LIN {X 0,Y 626.44,Z 347.198,A -85,B 0,C 180,E1 29853.409,E2 29853.409} C_VEL
LIN {X 0,Y 625.043,Z 344.117,A -85,B 0,C 180,E1 29853.056,E2 29853.056} C_VEL
LIN {X 0,Y 624.945,Z 343.42,A -85,B 0,C 180,E1 29852.768,E2 29852.768} C_VEL
LIN {X 0,Y 624.921,Z 343.391,A -85,B 0,C 180,E1 29849.587,E2 29849.587} C_VEL
LIN {X 0,Y 624.985,Z 343.634,A -85,B 0,C 180,E1 29846.589,E2 29846.589} C_VEL
LIN {X 0,Y 626.32,Z 346.962,A -85,B 0,C 180,E1 29846.03,E2 29846.03} C_VEL
LIN {X 0,Y 627.286,Z 348.589,A -85,B 0,C 180,E1 29845.758,E2 29845.758} C_VEL
LIN {X 0,Y 631.043,Z 356.586,A -85,B 0,C 180,E1 29844.666,E2 29844.666} C_VEL
LIN {X 0,Y 636.482,Z 369.43,A -85,B 0,C 180,E1 29843.235,E2 29843.235} C_VEL
LIN {X 0,Y 643.968,Z 387.871,A -85,B 0,C 180,E1 29841.491,E2 29841.491} C_VEL
LIN {X 0,Y 650.226,Z 398.532,A -85,B 0,C 180,E1 29840.459,E2 29840.459} C_VEL
LIN {X 0,Y 650.452,Z 412.85,A -85,B 0,C 180,E1 29839.657,E2 29839.657} C_VEL
LIN {X 0,Y 655.73,Z 440.789,A -85,B 0,C 180,E1 29838.782,E2 29838.782} C_VEL
LIN {X 0,Y 660.63,Z 462.04,A -85,B 0,C 180,E1 29838.099,E2 29838.099} C_VEL
LIN {X 0,Y 658.56,Z 625.386,A -85,B 0,C 180,E1 29835.964,E2 29835.964} C_VEL
LIN {X 0,Y 654.313,Z 847.674,A -85,B 0,C 180,E1 29832.989,E2 29832.989} C_VEL
LIN {X 0,Y 653.026,Z 907.79,A -85,B 0,C 180,E1 29832.173,E2 29832.173} C_VEL
LIN {X 0,Y 651.72,Z 936.587,A -85,B 0,C 180,E1 29831.618,E2 29831.618} C_VEL
LIN {X 0,Y 650.342,Z 959.946,A -85,B 0,C 180,E1 29831.02,E2 29831.02} C_VEL
LIN {X 0,Y 648.895,Z 981.108,A -85,B 0,C 180,E1 29830.358,E2 29830.358} C_VEL
LIN {X 0,Y 647.293,Z 1002.373,A -85,B 0,C 180,E1 29829.572,E2 29829.572} C_VEL
LIN {X 0,Y 645.185,Z 1027.649,A -85,B 0,C 180,E1 29828.479,E2 29828.479} C_VEL
LIN {X 0,Y 642.948,Z 1051.037,A -85,B 0,C 180,E1 29827.281,E2 29827.281} C_VEL
LIN {X 0,Y 640.981,Z 1070.815,A -85,B 0,C 180,E1 29826.132,E2 29826.132} C_VEL
LIN {X 0,Y 639.019,Z 1089.996,A -85,B 0,C 180,E1 29824.883,E2 29824.883} C_VEL
LIN {X 0,Y 636.733,Z 1111.873,A -85,B 0,C 180,E1 29823.287,E2 29823.287} C_VEL
LIN {X 0,Y 634.481,Z 1133.139,A -85,B 0,C 180,E1 29821.507,E2 29821.507} C_VEL
LIN {X 0,Y 632.771,Z 1149.796,A -85,B 0,C 180,E1 29819.956,E2 29819.956} C_VEL
LIN {X 0,Y 631.114,Z 1166.381,A -85,B 0,C 180,E1 29818.25,E2 29818.25} C_VEL
LIN {X 0,Y 629.253,Z 1185.743,A -85,B 0,C 180,E1 29816.012,E2 29816.012} C_VEL
LIN {X 0,Y 627.941,Z 1200.693,A -85,B 0,C 180,E1 29814.056,E2 29814.056} C_VEL
LIN {X 0,Y 626.836,Z 1214.647,A -85,B 0,C 180,E1 29812.015,E2 29812.015} C_VEL
LIN {X 0,Y 625.791,Z 1229.67,A -85,B 0,C 180,E1 29809.508,E2 29809.508} C_VEL
LIN {X 0,Y 625.132,Z 1240.614,A -85,B 0,C 180,E1 29807.403,E2 29807.403} C_VEL
LIN {X 0,Y 624.666,Z 1249.714,A -85,B 0,C 180,E1 29805.409,E2 29805.409} C_VEL
LIN {X 0,Y 624.334,Z 1258.281,A -85,B 0,C 180,E1 29803.239,E2 29803.239} C_VEL
LIN {X 0,Y 624.09,Z 1266.776,A -85,B 0,C 180,E1 29800.617,E2 29800.617} C_VEL
LIN {X 0,Y 623.98,Z 1272.734,A -85,B 0,C 180,E1 29798.292,E2 29798.292} C_VEL
LIN {X 0,Y 623.933,Z 1277.189,A -85,B 0,C 180,E1 29795.979,E2 29795.979} C_VEL
LIN {X 0,Y 623.912,Z 1280.336,A -85,B 0,C 180,E1 29793.491,E2 29793.491} C_VEL
LIN {X 0,Y 623.889,Z 1281.714,A -85,B 0,C 180,E1 29791.194,E2 29791.194} C_VEL
LIN {X 0,Y 623.864,Z 1281.827,A -85,B 0,C 180,E1 29789.265,E2 29789.265} C_VEL
LIN {X 0,Y 623.908,Z 1280.947,A -85,B 0,C 180,E1 29787.336,E2 29787.336} C_VEL
LIN {X 0,Y 623.916,Z 1278.899,A -85,B 0,C 180,E1 29785.22,E2 29785.22} C_VEL
LIN {X 0,Y 623.954,Z 1275.078,A -85,B 0,C 180,E1 29782.82,E2 29782.82} C_VEL
LIN {X 0,Y 623.985,Z 1269.837,A -85,B 0,C 180,E1 29780.5,E2 29780.5} C_VEL
LIN {X 0,Y 624.176,Z 1263.356,A -85,B 0,C 180,E1 29778.262,E2 29778.262} C_VEL
LIN {X 0,Y 624.361,Z 1256.514,A -85,B 0,C 180,E1 29776.29,E2 29776.29} C_VEL
LIN {X 0,Y 624.701,Z 1248.901,A -85,B 0,C 180,E1 29774.401,E2 29774.401} C_VEL
LIN {X 0,Y 625.202,Z 1239.22,A -85,B 0,C 180,E1 29772.31,E2 29772.31} C_VEL
LIN {X 0,Y 626.035,Z 1225.878,A -85,B 0,C 180,E1 29769.819,E2 29769.819} C_VEL
LIN {X 0,Y 626.999,Z 1212.519,A -85,B 0,C 180,E1 29767.66,E2 29767.66} C_VEL
LIN {X 0,Y 628.138,Z 1198.567,A -85,B 0,C 180,E1 29765.652,E2 29765.652} C_VEL
LIN {X 0,Y 629.787,Z 1180.067,A -85,B 0,C 180,E1 29763.301,E2 29763.301} C_VEL
LIN {X 0,Y 631.389,Z 1163.378,A -85,B 0,C 180,E1 29761.429,E2 29761.429} C_VEL
LIN {X 0,Y 633.123,Z 1146.246,A -85,B 0,C 180,E1 29759.697,E2 29759.697} C_VEL
LIN {X 0,Y 635.507,Z 1123.476,A -85,B 0,C 180,E1 29757.66,E2 29757.66} C_VEL
LIN {X 0,Y 637.417,Z 1105.296,A -85,B 0,C 180,E1 29756.22,E2 29756.22} C_VEL
LIN {X 0,Y 639.321,Z 1087.049,A -85,B 0,C 180,E1 29754.917,E2 29754.917} C_VEL
LIN {X 0,Y 641.405,Z 1066.751,A -85,B 0,C 180,E1 29753.619,E2 29753.619} C_VEL
LIN {X 0,Y 643.914,Z 1040.714,A -85,B 0,C 180,E1 29752.167,E2 29752.167} C_VEL
LIN {X 0,Y 645.879,Z 1018.721,A -85,B 0,C 180,E1 29751.116,E2 29751.116} C_VEL
LIN {X 0,Y 647.601,Z 998.037,A -85,B 0,C 180,E1 29750.256,E2 29750.256} C_VEL
LIN {X 0,Y 649.274,Z 975.928,A -85,B 0,C 180,E1 29749.468,E2 29749.468} C_VEL
LIN {X 0,Y 651.08,Z 948.454,A -85,B 0,C 180,E1 29748.665,E2 29748.665} C_VEL
LIN {X 0,Y 652.353,Z 923.49,A -85,B 0,C 180,E1 29748.107,E2 29748.107} C_VEL
LIN {X 0,Y 653.236,Z 900.801,A -85,B 0,C 180,E1 29747.723,E2 29747.723} C_VEL
LIN {X 0,Y 657.429,Z 682.384,A -85,B 0,C 180,E1 29744.806,E2 29744.806} C_VEL
LIN {X 0,Y 661.107,Z 486.103,A -85,B 0,C 180,E1 29742.148,E2 29742.148} C_VEL
LIN {X 0,Y 661.403,Z 460.724,A -85,B 0,C 180,E1 29741.783,E2 29741.783} C_VEL
LIN {X 0,Y 653.875,Z 423.501,A -85,B 0,C 180,E1 29740.419,E2 29740.419} C_VEL
LIN {X 0,Y 655.004,Z 402.248,A -85,B 0,C 180,E1 29739.014,E2 29739.014} C_VEL
LIN {X 0,Y 643.082,Z 378.276,A -85,B 0,C 180,E1 29735.996,E2 29735.996} C_VEL
LIN {X 0,Y 636.424,Z 365.479,A -85,B 0,C 180,E1 29734.226,E2 29734.226} C_VEL
LIN {X 0,Y 631.891,Z 356.934,A -85,B 0,C 180,E1 29732.98,E2 29732.98} C_VEL
LIN {X 0,Y 629.323,Z 352.257,A -85,B 0,C 180,E1 29732.266,E2 29732.266} C_VEL
LIN {X 0,Y 626.8,Z 347.598,A -85,B 0,C 180,E1 29731.55,E2 29731.55} C_VEL
LIN {X 0,Y 625.074,Z 344.123,A -85,B 0,C 180,E1 29731.003,E2 29731.003} C_VEL
LIN {X 0,Y 624.943,Z 343.458,A -85,B 0,C 180,E1 29730.776,E2 29730.776} C_VEL
LIN {X 0,Y 624.946,Z 343.386,A -85,B 0,C 180,E1 29727.645,E2 29727.645} C_VEL
LIN {X 0,Y 624.927,Z 343.382,A -85,B 0,C 180,E1 29724.482,E2 29724.482} C_VEL
LIN {X 0,Y 624.945,Z 343.377,A -85,B 0,C 180,E1 29721.383,E2 29721.383} C_VEL
LIN {X 0,Y 624.924,Z 343.376,A -85,B 0,C 180,E1 29718.277,E2 29718.277} C_VEL
LIN {X 0,Y 624.945,Z 343.375,A -85,B 0,C 180,E1 29715.212,E2 29715.212} C_VEL
LIN {X 0,Y 624.921,Z 343.375,A -85,B 0,C 180,E1 29712.099,E2 29712.099} C_VEL
LIN {X 0,Y 624.947,Z 343.377,A -85,B 0,C 180,E1 29709.021,E2 29709.021} C_VEL
LIN {X 0,Y 624.919,Z 343.378,A -85,B 0,C 180,E1 29705.97,E2 29705.97} C_VEL
LIN {X 0,Y 624.949,Z 343.384,A -85,B 0,C 180,E1 29702.843,E2 29702.843} C_VEL
LIN {X 0,Y 624.916,Z 343.386,A -85,B 0,C 180,E1 29699.725,E2 29699.725} C_VEL
LIN {X 0,Y 624.949,Z 343.382,A -85,B 0,C 180,E1 29696.606,E2 29696.606} C_VEL
LIN {X 0,Y 624.912,Z 343.384,A -85,B 0,C 180,E1 29693.477,E2 29693.477} C_VEL
LIN {X 0,Y 624.952,Z 343.382,A -85,B 0,C 180,E1 29690.422,E2 29690.422} C_VEL
LIN {X 0,Y 624.911,Z 343.386,A -85,B 0,C 180,E1 29687.337,E2 29687.337} C_VEL
LIN {X 0,Y 624.956,Z 343.382,A -85,B 0,C 180,E1 29684.312,E2 29684.312} C_VEL
LIN {X 0,Y 624.91,Z 343.387,A -85,B 0,C 180,E1 29681.239,E2 29681.239} C_VEL
LIN {X 0,Y 624.956,Z 343.381,A -85,B 0,C 180,E1 29678.211,E2 29678.211} C_VEL
LIN {X 0,Y 624.911,Z 343.387,A -85,B 0,C 180,E1 29675.114,E2 29675.114} C_VEL
LIN {X 0,Y 624.957,Z 343.381,A -85,B 0,C 180,E1 29672.025,E2 29672.025} C_VEL
LIN {X 0,Y 624.905,Z 343.387,A -85,B 0,C 180,E1 29668.873,E2 29668.873} C_VEL
LIN {X 0,Y 624.954,Z 343.381,A -85,B 0,C 180,E1 29665.808,E2 29665.808} C_VEL
LIN {X 0,Y 624.9,Z 343.388,A -85,B 0,C 180,E1 29662.668,E2 29662.668} C_VEL
LIN {X 0,Y 624.942,Z 343.381,A -85,B 0,C 180,E1 29659.73,E2 29659.73} C_VEL
LIN {X 0,Y 624.901,Z 343.388,A -85,B 0,C 180,E1 29656.525,E2 29656.525} C_VEL
LIN {X 0,Y 624.938,Z 343.381,A -85,B 0,C 180,E1 29653.548,E2 29653.548} C_VEL
LIN {X 0,Y 624.899,Z 343.389,A -85,B 0,C 180,E1 29650.391,E2 29650.391} C_VEL
LIN {X 0,Y 624.889,Z 343.386,A -85,B 0,C 180,E1 29648.108,E2 29648.108} C_VEL
LIN {X 0,Y 623.91,Z 343.51,A -85,B 0,C 180,E1 29647.401,E2 29647.401} C_VEL
LIN {X 0,Y 617.551,Z 344.298,A -85,B 0,C 180,E1 29645.42,E2 29645.42} C_VEL
LIN {X 0,Y 617.016,Z 344.367,A -85,B 0,C 180,E1 29644.905,E2 29644.905} C_VEL
LIN {X 0,Y 616.947,Z 344.374,A -85,B 0,C 180,E1 29641.869,E2 29641.869} C_VEL
LIN {X 0,Y 617.019,Z 344.364,A -85,B 0,C 180,E1 29638.875,E2 29638.875} C_VEL
LIN {X 0,Y 616.947,Z 344.375,A -85,B 0,C 180,E1 29635.847,E2 29635.847} C_VEL
LIN {X 0,Y 616.991,Z 344.365,A -85,B 0,C 180,E1 29632.888,E2 29632.888} C_VEL
LIN {X 0,Y 616.949,Z 344.379,A -85,B 0,C 180,E1 29629.799,E2 29629.799} C_VEL
LIN {X 0,Y 616.959,Z 344.374,A -85,B 0,C 180,E1 29626.961,E2 29626.961} C_VEL
LIN {X 0,Y 616.952,Z 344.379,A -85,B 0,C 180,E1 29623.687,E2 29623.687} C_VEL
LIN {X 0,Y 616.944,Z 344.379,A -85,B 0,C 180,E1 29620.931,E2 29620.931} C_VEL
LIN {X 0,Y 616.968,Z 344.374,A -85,B 0,C 180,E1 29617.73,E2 29617.73} C_VEL
LIN {X 0,Y 616.931,Z 344.373,A -85,B 0,C 180,E1 29614.928,E2 29614.928} C_VEL
LIN {X 0,Y 617.003,Z 344.374,A -85,B 0,C 180,E1 29611.857,E2 29611.857} C_VEL
LIN {X 0,Y 616.929,Z 344.382,A -85,B 0,C 180,E1 29608.979,E2 29608.979} C_VEL
LIN {X 0,Y 616.97,Z 344.359,A -85,B 0,C 180,E1 29606.097,E2 29606.097} C_VEL
LIN {X 0,Y 616.931,Z 344.354,A -85,B 0,C 180,E1 29603.018,E2 29603.018} C_VEL
LIN {X 0,Y 616.926,Z 344.371,A -85,B 0,C 180,E1 29600.39,E2 29600.39} C_VEL
LIN {X 0,Y 617.025,Z 344.571,A -85,B 0,C 180,E1 29597.601,E2 29597.601} C_VEL
LIN {X 0,Y 617.381,Z 346.03,A -85,B 0,C 180,E1 29597.395,E2 29597.395} C_VEL
LIN {X 0,Y 619.284,Z 349.081,A -85,B 0,C 180,E1 29597.102,E2 29597.102} C_VEL
LIN {X 0,Y 621.278,Z 350.95,A -85,B 0,C 180,E1 29596.83,E2 29596.83} C_VEL
LIN {X 0,Y 623.786,Z 354.703,A -85,B 0,C 180,E1 29596.466,E2 29596.466} C_VEL
LIN {X 0,Y 625.81,Z 356.86,A -85,B 0,C 180,E1 29596.193,E2 29596.193} C_VEL
LIN {X 0,Y 629.122,Z 361.131,A -85,B 0,C 180,E1 29595.739,E2 29595.739} C_VEL
LIN {X 0,Y 633.273,Z 366.632,A -85,B 0,C 180,E1 29595.18,E2 29595.18} C_VEL
LIN {X 0,Y 649.293,Z 388.598,A -85,B 0,C 180,E1 29593.148,E2 29593.148} C_VEL
LIN {X 0,Y 654.652,Z 396.391,A -85,B 0,C 180,E1 29592.508,E2 29592.508} C_VEL
LIN {X 0,Y 650.14,Z 613.265,A -85,B 0,C 180,E1 29589.557,E2 29589.557} C_VEL
LIN {X 0,Y 647.14,Z 757.621,A -85,B 0,C 180,E1 29587.612,E2 29587.612} C_VEL
LIN {X 0,Y 645.877,Z 783.784,A -85,B 0,C 180,E1 29587.113,E2 29587.113} C_VEL
LIN {X 0,Y 644.236,Z 810.568,A -85,B 0,C 180,E1 29586.432,E2 29586.432} C_VEL
LIN {X 0,Y 642.332,Z 836.613,A -85,B 0,C 180,E1 29585.595,E2 29585.595} C_VEL
LIN {X 0,Y 640.2,Z 862.261,A -85,B 0,C 180,E1 29584.589,E2 29584.589} C_VEL
LIN {X 0,Y 637.88,Z 886.313,A -85,B 0,C 180,E1 29583.466,E2 29583.466} C_VEL
LIN {X 0,Y 635.242,Z 911.914,A -85,B 0,C 180,E1 29582.073,E2 29582.073} C_VEL
LIN {X 0,Y 632.667,Z 935.913,A -85,B 0,C 180,E1 29580.555,E2 29580.555} C_VEL
LIN {X 0,Y 630.387,Z 956.418,A -85,B 0,C 180,E1 29579.076,E2 29579.076} C_VEL
LIN {X 0,Y 627.823,Z 978.962,A -85,B 0,C 180,E1 29577.237,E2 29577.237} C_VEL
LIN {X 0,Y 625.456,Z 1000.26,A -85,B 0,C 180,E1 29575.257,E2 29575.257} C_VEL
LIN {X 0,Y 623.342,Z 1020.045,A -85,B 0,C 180,E1 29573.172,E2 29573.172} C_VEL
LIN {X 0,Y 621.513,Z 1038.014,A -85,B 0,C 180,E1 29571.021,E2 29571.021} C_VEL
LIN {X 0,Y 619.972,Z 1054.397,A -85,B 0,C 180,E1 29568.807,E2 29568.807} C_VEL
LIN {X 0,Y 618.665,Z 1070.031,A -85,B 0,C 180,E1 29566.391,E2 29566.391} C_VEL
LIN {X 0,Y 617.768,Z 1082.311,A -85,B 0,C 180,E1 29564.235,E2 29564.235} C_VEL
LIN {X 0,Y 617.026,Z 1093.97,A -85,B 0,C 180,E1 29561.886,E2 29561.886} C_VEL
LIN {X 0,Y 616.526,Z 1104.735,A -85,B 0,C 180,E1 29559.322,E2 29559.322} C_VEL
LIN {X 0,Y 616.199,Z 1112.49,A -85,B 0,C 180,E1 29557.131,E2 29557.131} C_VEL
LIN {X 0,Y 616.046,Z 1119.459,A -85,B 0,C 180,E1 29554.73,E2 29554.73} C_VEL
LIN {X 0,Y 615.934,Z 1124.777,A -85,B 0,C 180,E1 29552.393,E2 29552.393} C_VEL
LIN {X 0,Y 615.929,Z 1128.644,A -85,B 0,C 180,E1 29550,E2 29550} C_VEL
LIN {X 0,Y 615.888,Z 1131.051,A -85,B 0,C 180,E1 29547.574,E2 29547.574} C_VEL
LIN {X 0,Y 615.901,Z 1131.941,A -85,B 0,C 180,E1 29545.276,E2 29545.276} C_VEL
LIN {X 0,Y 615.865,Z 1131.328,A -85,B 0,C 180,E1 29542.756,E2 29542.756} C_VEL
LIN {X 0,Y 615.915,Z 1129.328,A -85,B 0,C 180,E1 29540.428,E2 29540.428} C_VEL
LIN {X 0,Y 615.948,Z 1125.598,A -85,B 0,C 180,E1 29537.962,E2 29537.962} C_VEL
LIN {X 0,Y 616.037,Z 1120.12,A -85,B 0,C 180,E1 29535.438,E2 29535.438} C_VEL
LIN {X 0,Y 616.205,Z 1113.002,A -85,B 0,C 180,E1 29532.94,E2 29532.94} C_VEL
LIN {X 0,Y 616.487,Z 1105.704,A -85,B 0,C 180,E1 29530.844,E2 29530.844} C_VEL
LIN {X 0,Y 616.969,Z 1095.624,A -85,B 0,C 180,E1 29528.387,E2 29528.387} C_VEL
LIN {X 0,Y 617.681,Z 1083.75,A -85,B 0,C 180,E1 29525.947,E2 29525.947} C_VEL
LIN {X 0,Y 618.592,Z 1071.179,A -85,B 0,C 180,E1 29523.707,E2 29523.707} C_VEL
LIN {X 0,Y 619.811,Z 1056.349,A -85,B 0,C 180,E1 29521.387,E2 29521.387} C_VEL
LIN {X 0,Y 621.372,Z 1039.468,A -85,B 0,C 180,E1 29519.078,E2 29519.078} C_VEL
LIN {X 0,Y 623.025,Z 1022.847,A -85,B 0,C 180,E1 29517.056,E2 29517.056} C_VEL
LIN {X 0,Y 625.243,Z 1002.388,A -85,B 0,C 180,E1 29514.862,E2 29514.862} C_VEL
LIN {X 0,Y 627.462,Z 982.118,A -85,B 0,C 180,E1 29512.952,E2 29512.952} C_VEL
LIN {X 0,Y 630.054,Z 959.257,A -85,B 0,C 180,E1 29511.053,E2 29511.053} C_VEL
LIN {X 0,Y 632.554,Z 937.101,A -85,B 0,C 180,E1 29509.434,E2 29509.434} C_VEL
LIN {X 0,Y 635.206,Z 912.533,A -85,B 0,C 180,E1 29507.869,E2 29507.869} C_VEL
LIN {X 0,Y 637.696,Z 888.159,A -85,B 0,C 180,E1 29506.535,E2 29506.535} C_VEL
LIN {X 0,Y 640.033,Z 863.672,A -85,B 0,C 180,E1 29505.386,E2 29505.386} C_VEL
LIN {X 0,Y 642.204,Z 838.307,A -85,B 0,C 180,E1 29504.374,E2 29504.374} C_VEL
LIN {X 0,Y 644.064,Z 812.942,A -85,B 0,C 180,E1 29503.547,E2 29503.547} C_VEL
LIN {X 0,Y 645.778,Z 785.479,A -85,B 0,C 180,E1 29502.836,E2 29502.836} C_VEL
LIN {X 0,Y 647.033,Z 760.107,A -85,B 0,C 180,E1 29502.34,E2 29502.34} C_VEL
LIN {X 0,Y 648.218,Z 710.458,A -85,B 0,C 180,E1 29501.653,E2 29501.653} C_VEL
LIN {X 0,Y 652.209,Z 504.112,A -85,B 0,C 180,E1 29498.893,E2 29498.893} C_VEL
LIN {X 0,Y 654.095,Z 395.736,A -85,B 0,C 180,E1 29497.413,E2 29497.413} C_VEL
LIN {X 0,Y 639.586,Z 375.63,A -85,B 0,C 180,E1 29495.674,E2 29495.674} C_VEL
LIN {X 0,Y 632.819,Z 366.077,A -85,B 0,C 180,E1 29494.712,E2 29494.712} C_VEL
LIN {X 0,Y 629.184,Z 361.107,A -85,B 0,C 180,E1 29494.145,E2 29494.145} C_VEL
LIN {X 0,Y 626.323,Z 356.874,A -85,B 0,C 180,E1 29493.641,E2 29493.641} C_VEL
LIN {X 0,Y 622.996,Z 353.334,A -85,B 0,C 180,E1 29493.05,E2 29493.05} C_VEL
LIN {X 0,Y 621.527,Z 350.643,A -85,B 0,C 180,E1 29492.726,E2 29492.726} C_VEL
LIN {X 0,Y 618.454,Z 348.053,A -85,B 0,C 180,E1 29492.073,E2 29492.073} C_VEL
LIN {X 0,Y 617.11,Z 345.139,A -85,B 0,C 180,E1 29491.618,E2 29491.618} C_VEL
LIN {X 0,Y 616.977,Z 344.413,A -85,B 0,C 180,E1 29491.228,E2 29491.228} C_VEL
LIN {X 0,Y 617.014,Z 344.376,A -85,B 0,C 180,E1 29488.11,E2 29488.11} C_VEL
LIN {X 0,Y 617.06,Z 344.812,A -85,B 0,C 180,E1 29487.674,E2 29487.674} C_VEL
LIN {X 0,Y 618.456,Z 348.097,A -85,B 0,C 180,E1 29486.986,E2 29486.986} C_VEL
LIN {X 0,Y 619.613,Z 349.9,A -85,B 0,C 180,E1 29486.613,E2 29486.613} C_VEL
LIN {X 0,Y 622.023,Z 355.115,A -85,B 0,C 180,E1 29485.763,E2 29485.763} C_VEL
LIN {X 0,Y 625.43,Z 362.431,A -85,B 0,C 180,E1 29484.75,E2 29484.75} C_VEL
LIN {X 0,Y 630.385,Z 374.351,A -85,B 0,C 180,E1 29483.388,E2 29483.388} C_VEL
LIN {X 0,Y 637.71,Z 392.65,A -85,B 0,C 180,E1 29481.618,E2 29481.618} C_VEL
LIN {X 0,Y 643.308,Z 402.169,A -85,B 0,C 180,E1 29480.671,E2 29480.671} C_VEL
LIN {X 0,Y 643.497,Z 407.96,A -85,B 0,C 180,E1 29480.361,E2 29480.361} C_VEL
LIN {X 0,Y 650.125,Z 444.426,A -85,B 0,C 180,E1 29479.171,E2 29479.171} C_VEL
LIN {X 0,Y 654.533,Z 463.978,A -85,B 0,C 180,E1 29478.531,E2 29478.531} C_VEL
LIN {X 0,Y 652.544,Z 612.386,A -85,B 0,C 180,E1 29476.579,E2 29476.579} C_VEL
LIN {X 0,Y 651.281,Z 707.38,A -85,B 0,C 180,E1 29475.355,E2 29475.355} C_VEL
LIN {X 0,Y 647.193,Z 904.317,A -85,B 0,C 180,E1 29472.703,E2 29472.703} C_VEL
LIN {X 0,Y 646.07,Z 930.59,A -85,B 0,C 180,E1 29472.23,E2 29472.23} C_VEL
LIN {X 0,Y 644.42,Z 957.585,A -85,B 0,C 180,E1 29471.56,E2 29471.56} C_VEL
LIN {X 0,Y 642.878,Z 979.062,A -85,B 0,C 180,E1 29470.896,E2 29470.896} C_VEL
LIN {X 0,Y 641.217,Z 999.571,A -85,B 0,C 180,E1 29470.15,E2 29470.15} C_VEL
LIN {X 0,Y 639.315,Z 1020.973,A -85,B 0,C 180,E1 29469.244,E2 29469.244} C_VEL
LIN {X 0,Y 636.881,Z 1046.532,A -85,B 0,C 180,E1 29467.983,E2 29467.983} C_VEL
LIN {X 0,Y 634.478,Z 1069.189,A -85,B 0,C 180,E1 29466.674,E2 29466.674} C_VEL
LIN {X 0,Y 632.44,Z 1087.789,A -85,B 0,C 180,E1 29465.466,E2 29465.466} C_VEL
LIN {X 0,Y 630.425,Z 1105.899,A -85,B 0,C 180,E1 29464.156,E2 29464.156} C_VEL
LIN {X 0,Y 628.076,Z 1126.929,A -85,B 0,C 180,E1 29462.461,E2 29462.461} C_VEL
LIN {X 0,Y 625.702,Z 1147.856,A -85,B 0,C 180,E1 29460.532,E2 29460.532} C_VEL
LIN {X 0,Y 623.918,Z 1164.304,A -85,B 0,C 180,E1 29458.841,E2 29458.841} C_VEL
LIN {X 0,Y 622.05,Z 1182.6,A -85,B 0,C 180,E1 29456.748,E2 29456.748} C_VEL
LIN {X 0,Y 620.377,Z 1199.99,A -85,B 0,C 180,E1 29454.47,E2 29454.47} C_VEL
LIN {X 0,Y 619.154,Z 1214.01,A -85,B 0,C 180,E1 29452.403,E2 29452.403} C_VEL
LIN {X 0,Y 618.004,Z 1229.149,A -85,B 0,C 180,E1 29449.862,E2 29449.862} C_VEL
LIN {X 0,Y 617.245,Z 1240.616,A -85,B 0,C 180,E1 29447.633,E2 29447.633} C_VEL
LIN {X 0,Y 616.719,Z 1250.117,A -85,B 0,C 180,E1 29445.516,E2 29445.516} C_VEL
LIN {X 0,Y 616.351,Z 1259.339,A -85,B 0,C 180,E1 29443.127,E2 29443.127} C_VEL
LIN {X 0,Y 616.099,Z 1267.033,A -85,B 0,C 180,E1 29440.662,E2 29440.662} C_VEL
LIN {X 0,Y 615.994,Z 1272.731,A -85,B 0,C 180,E1 29438.4,E2 29438.4} C_VEL
LIN {X 0,Y 615.934,Z 1277.337,A -85,B 0,C 180,E1 29435.963,E2 29435.963} C_VEL
LIN {X 0,Y 615.911,Z 1280.404,A -85,B 0,C 180,E1 29433.444,E2 29433.444} C_VEL
LIN {X 0,Y 615.89,Z 1281.714,A -85,B 0,C 180,E1 29431.209,E2 29431.209} C_VEL
LIN {X 0,Y 615.864,Z 1281.827,A -85,B 0,C 180,E1 29429.256,E2 29429.256} C_VEL
LIN {X 0,Y 615.908,Z 1280.947,A -85,B 0,C 180,E1 29427.302,E2 29427.302} C_VEL
LIN {X 0,Y 615.916,Z 1279.009,A -85,B 0,C 180,E1 29425.251,E2 29425.251} C_VEL
LIN {X 0,Y 615.956,Z 1275.25,A -85,B 0,C 180,E1 29422.82,E2 29422.82} C_VEL
LIN {X 0,Y 616.001,Z 1269.837,A -85,B 0,C 180,E1 29420.376,E2 29420.376} C_VEL
LIN {X 0,Y 616.197,Z 1263.306,A -85,B 0,C 180,E1 29418.092,E2 29418.092} C_VEL
LIN {X 0,Y 616.406,Z 1256.513,A -85,B 0,C 180,E1 29416.109,E2 29416.109} C_VEL
LIN {X 0,Y 616.785,Z 1248.902,A -85,B 0,C 180,E1 29414.196,E2 29414.196} C_VEL
LIN {X 0,Y 617.314,Z 1239.222,A -85,B 0,C 180,E1 29412.076,E2 29412.076} C_VEL
LIN {X 0,Y 618.227,Z 1225.876,A -85,B 0,C 180,E1 29409.553,E2 29409.553} C_VEL
LIN {X 0,Y 619.255,Z 1212.741,A -85,B 0,C 180,E1 29407.401,E2 29407.401} C_VEL
LIN {X 0,Y 620.507,Z 1198.569,A -85,B 0,C 180,E1 29405.333,E2 29405.333} C_VEL
LIN {X 0,Y 622.307,Z 1180.065,A -85,B 0,C 180,E1 29402.954,E2 29402.954} C_VEL
LIN {X 0,Y 624.01,Z 1163.377,A -85,B 0,C 180,E1 29401.059,E2 29401.059} C_VEL
LIN {X 0,Y 625.88,Z 1146.243,A -85,B 0,C 180,E1 29399.308,E2 29399.308} C_VEL
LIN {X 0,Y 628.451,Z 1123.477,A -85,B 0,C 180,E1 29397.252,E2 29397.252} C_VEL
LIN {X 0,Y 630.495,Z 1105.226,A -85,B 0,C 180,E1 29395.793,E2 29395.793} C_VEL
LIN {X 0,Y 632.487,Z 1087.352,A -85,B 0,C 180,E1 29394.504,E2 29394.504} C_VEL
LIN {X 0,Y 634.565,Z 1068.371,A -85,B 0,C 180,E1 29393.275,E2 29393.275} C_VEL
LIN {X 0,Y 637.07,Z 1044.692,A -85,B 0,C 180,E1 29391.916,E2 29391.916} C_VEL
LIN {X 0,Y 639.415,Z 1019.848,A -85,B 0,C 180,E1 29390.705,E2 29390.705} C_VEL
LIN {X 0,Y 641.277,Z 998.805,A -85,B 0,C 180,E1 29389.82,E2 29389.82} C_VEL
LIN {X 0,Y 643.002,Z 977.405,A -85,B 0,C 180,E1 29389.047,E2 29389.047} C_VEL
LIN {X 0,Y 644.867,Z 951.337,A -85,B 0,C 180,E1 29388.264,E2 29388.264} C_VEL
LIN {X 0,Y 646.329,Z 924.602,A -85,B 0,C 180,E1 29387.653,E2 29387.653} C_VEL
LIN {X 0,Y 647.275,Z 901.947,A -85,B 0,C 180,E1 29387.262,E2 29387.262} C_VEL
LIN {X 0,Y 651.587,Z 691.755,A -85,B 0,C 180,E1 29384.433,E2 29384.433} C_VEL
LIN {X 0,Y 655.567,Z 485.945,A -85,B 0,C 180,E1 29381.639,E2 29381.639} C_VEL
LIN {X 0,Y 655.86,Z 462.778,A -85,B 0,C 180,E1 29381.303,E2 29381.303} C_VEL
LIN {X 0,Y 647.915,Z 422.962,A -85,B 0,C 180,E1 29379.825,E2 29379.825} C_VEL
LIN {X 0,Y 648.846,Z 406.53,A -85,B 0,C 180,E1 29378.731,E2 29378.731} C_VEL
LIN {X 0,Y 636.194,Z 380.875,A -85,B 0,C 180,E1 29375.447,E2 29375.447} C_VEL
LIN {X 0,Y 626.696,Z 362.853,A -85,B 0,C 180,E1 29372.852,E2 29372.852} C_VEL
LIN {X 0,Y 621.626,Z 353.526,A -85,B 0,C 180,E1 29371.41,E2 29371.41} C_VEL
LIN {X 0,Y 619.174,Z 348.965,A -85,B 0,C 180,E1 29370.684,E2 29370.684} C_VEL
LIN {X 0,Y 617.266,Z 345.616,A -85,B 0,C 180,E1 29370.118,E2 29370.118} C_VEL
LIN {X 0,Y 617.035,Z 344.519,A -85,B 0,C 180,E1 29369.895,E2 29369.895} C_VEL
LIN {X 0,Y 616.994,Z 344.365,A -85,B 0,C 180,E1 29366.673,E2 29366.673} C_VEL
LIN {X 0,Y 617.005,Z 344.362,A -85,B 0,C 180,E1 29363.494,E2 29363.494} C_VEL
LIN {X 0,Y 616.988,Z 344.369,A -85,B 0,C 180,E1 29360.391,E2 29360.391} C_VEL
LIN {X 0,Y 617.006,Z 344.367,A -85,B 0,C 180,E1 29357.251,E2 29357.251} C_VEL
LIN {X 0,Y 616.985,Z 344.375,A -85,B 0,C 180,E1 29354.165,E2 29354.165} C_VEL
LIN {X 0,Y 617.008,Z 344.365,A -85,B 0,C 180,E1 29351.024,E2 29351.024} C_VEL
LIN {X 0,Y 616.98,Z 344.372,A -85,B 0,C 180,E1 29347.918,E2 29347.918} C_VEL
LIN {X 0,Y 617.008,Z 344.36,A -85,B 0,C 180,E1 29344.834,E2 29344.834} C_VEL
LIN {X 0,Y 616.977,Z 344.363,A -85,B 0,C 180,E1 29341.765,E2 29341.765} C_VEL
LIN {X 0,Y 617.011,Z 344.371,A -85,B 0,C 180,E1 29338.7,E2 29338.7} C_VEL
LIN {X 0,Y 616.975,Z 344.372,A -85,B 0,C 180,E1 29335.538,E2 29335.538} C_VEL
LIN {X 0,Y 617.013,Z 344.371,A -85,B 0,C 180,E1 29332.457,E2 29332.457} C_VEL
LIN {X 0,Y 616.972,Z 344.374,A -85,B 0,C 180,E1 29329.353,E2 29329.353} C_VEL
LIN {X 0,Y 617.014,Z 344.373,A -85,B 0,C 180,E1 29326.219,E2 29326.219} C_VEL
LIN {X 0,Y 616.968,Z 344.367,A -85,B 0,C 180,E1 29323.136,E2 29323.136} C_VEL
LIN {X 0,Y 617.015,Z 344.369,A -85,B 0,C 180,E1 29320.005,E2 29320.005} C_VEL
LIN {X 0,Y 616.966,Z 344.368,A -85,B 0,C 180,E1 29317.002,E2 29317.002} C_VEL
LIN {X 0,Y 617.017,Z 344.369,A -85,B 0,C 180,E1 29313.865,E2 29313.865} C_VEL
LIN {X 0,Y 616.965,Z 344.368,A -85,B 0,C 180,E1 29310.802,E2 29310.802} C_VEL
LIN {X 0,Y 617.016,Z 344.371,A -85,B 0,C 180,E1 29307.769,E2 29307.769} C_VEL
LIN {X 0,Y 616.96,Z 344.37,A -85,B 0,C 180,E1 29304.649,E2 29304.649} C_VEL
LIN {X 0,Y 617.016,Z 344.372,A -85,B 0,C 180,E1 29301.635,E2 29301.635} C_VEL
LIN {X 0,Y 616.962,Z 344.372,A -85,B 0,C 180,E1 29298.606,E2 29298.606} C_VEL
LIN {X 0,Y 617.003,Z 344.373,A -85,B 0,C 180,E1 29295.566,E2 29295.566} C_VEL
LIN {X 0,Y 616.957,Z 344.373,A -85,B 0,C 180,E1 29292.391,E2 29292.391} C_VEL
LIN {X 0,Y 616.986,Z 344.374,A -85,B 0,C 180,E1 29289.519,E2 29289.519} C_VEL
LIN {X 0,Y 616.963,Z 344.374,A -85,B 0,C 180,E1 29286.344,E2 29286.344} C_VEL
LIN {X 0,Y 617.016,Z 344.367,A -85,B 0,C 180,E1 29284.905,E2 29284.905} C_VEL
LIN {X 0,Y 616.007,Z 344.499,A -85,B 0,C 180,E1 29284.19,E2 29284.19} C_VEL
LIN {X 0,Y 609.538,Z 345.298,A -85,B 0,C 180,E1 29282.184,E2 29282.184} C_VEL
LIN {X 0,Y 609.014,Z 345.362,A -85,B 0,C 180,E1 29281.661,E2 29281.661} C_VEL
LIN {X 0,Y 609.065,Z 345.359,A -85,B 0,C 180,E1 29278.537,E2 29278.537} C_VEL
LIN {X 0,Y 609.008,Z 345.363,A -85,B 0,C 180,E1 29275.582,E2 29275.582} C_VEL
LIN {X 0,Y 609.073,Z 345.359,A -85,B 0,C 180,E1 29272.443,E2 29272.443} C_VEL
LIN {X 0,Y 609.002,Z 345.367,A -85,B 0,C 180,E1 29269.469,E2 29269.469} C_VEL
LIN {X 0,Y 609.078,Z 345.364,A -85,B 0,C 180,E1 29266.401,E2 29266.401} C_VEL
LIN {X 0,Y 608.999,Z 345.367,A -85,B 0,C 180,E1 29263.385,E2 29263.385} C_VEL
LIN {X 0,Y 609.058,Z 345.363,A -85,B 0,C 180,E1 29260.404,E2 29260.404} C_VEL
LIN {X 0,Y 608.998,Z 345.364,A -85,B 0,C 180,E1 29257.358,E2 29257.358} C_VEL
LIN {X 0,Y 609.009,Z 345.361,A -85,B 0,C 180,E1 29254.614,E2 29254.614} C_VEL
LIN {X 0,Y 609.004,Z 345.37,A -85,B 0,C 180,E1 29251.317,E2 29251.317} C_VEL
LIN {X 0,Y 608.991,Z 345.37,A -85,B 0,C 180,E1 29248.683,E2 29248.683} C_VEL
LIN {X 0,Y 609.048,Z 345.357,A -85,B 0,C 180,E1 29245.575,E2 29245.575} C_VEL
LIN {X 0,Y 608.981,Z 345.344,A -85,B 0,C 180,E1 29242.621,E2 29242.621} C_VEL
LIN {X 0,Y 609.058,Z 345.334,A -85,B 0,C 180,E1 29239.596,E2 29239.596} C_VEL
LIN {X 0,Y 609.021,Z 345.637,A -85,B 0,C 180,E1 29238.542,E2 29238.542} C_VEL
LIN {X 0,Y 609.464,Z 347.254,A -85,B 0,C 180,E1 29238.334,E2 29238.334} C_VEL
LIN {X 0,Y 611.52,Z 350.248,A -85,B 0,C 180,E1 29238.015,E2 29238.015} C_VEL
LIN {X 0,Y 613.388,Z 351.861,A -85,B 0,C 180,E1 29237.754,E2 29237.754} C_VEL
LIN {X 0,Y 615.79,Z 355.603,A -85,B 0,C 180,E1 29237.391,E2 29237.391} C_VEL
LIN {X 0,Y 617.889,Z 357.873,A -85,B 0,C 180,E1 29237.096,E2 29237.096} C_VEL
LIN {X 0,Y 621.22,Z 362.173,A -85,B 0,C 180,E1 29236.622,E2 29236.622} C_VEL
LIN {X 0,Y 627.34,Z 370.335,A -85,B 0,C 180,E1 29235.768,E2 29235.768} C_VEL
LIN {X 0,Y 635.082,Z 380.613,A -85,B 0,C 180,E1 29234.733,E2 29234.733} C_VEL
LIN {X 0,Y 648.004,Z 398.521,A -85,B 0,C 180,E1 29233.114,E2 29233.114} C_VEL
LIN {X 0,Y 649.129,Z 400.484,A -85,B 0,C 180,E1 29232.972,E2 29232.972} C_VEL
LIN {X 0,Y 644.343,Z 616.732,A -85,B 0,C 180,E1 29230.009,E2 29230.009} C_VEL
LIN {X 0,Y 641.258,Z 757.495,A -85,B 0,C 180,E1 29228.1,E2 29228.1} C_VEL
LIN {X 0,Y 639.917,Z 783.86,A -85,B 0,C 180,E1 29227.595,E2 29227.595} C_VEL
LIN {X 0,Y 638.189,Z 810.616,A -85,B 0,C 180,E1 29226.911,E2 29226.911} C_VEL
LIN {X 0,Y 636.195,Z 836.44,A -85,B 0,C 180,E1 29226.079,E2 29226.079} C_VEL
LIN {X 0,Y 633.964,Z 861.802,A -85,B 0,C 180,E1 29225.08,E2 29225.08} C_VEL
LIN {X 0,Y 631.6,Z 885.086,A -85,B 0,C 180,E1 29223.991,E2 29223.991} C_VEL
LIN {X 0,Y 629.147,Z 907.969,A -85,B 0,C 180,E1 29222.761,E2 29222.761} C_VEL
LIN {X 0,Y 626.297,Z 932.686,A -85,B 0,C 180,E1 29221.222,E2 29221.222} C_VEL
LIN {X 0,Y 623.635,Z 955.073,A -85,B 0,C 180,E1 29219.609,E2 29219.609} C_VEL
LIN {X 0,Y 620.964,Z 977.32,A -85,B 0,C 180,E1 29217.793,E2 29217.793} C_VEL
LIN {X 0,Y 618.414,Z 998.547,A -85,B 0,C 180,E1 29215.822,E2 29215.822} C_VEL
LIN {X 0,Y 616.223,Z 1017.746,A -85,B 0,C 180,E1 29213.799,E2 29213.799} C_VEL
LIN {X 0,Y 614.109,Z 1036.575,A -85,B 0,C 180,E1 29211.551,E2 29211.551} C_VEL
LIN {X 0,Y 612.394,Z 1053.696,A -85,B 0,C 180,E1 29209.225,E2 29209.225} C_VEL
LIN {X 0,Y 610.99,Z 1069.077,A -85,B 0,C 180,E1 29206.839,E2 29206.839} C_VEL
LIN {X 0,Y 609.982,Z 1081.477,A -85,B 0,C 180,E1 29204.651,E2 29204.651} C_VEL
LIN {X 0,Y 609.193,Z 1093.131,A -85,B 0,C 180,E1 29202.295,E2 29202.295} C_VEL
LIN {X 0,Y 608.619,Z 1103.955,A -85,B 0,C 180,E1 29199.724,E2 29199.724} C_VEL
LIN {X 0,Y 608.243,Z 1112.025,A -85,B 0,C 180,E1 29197.44,E2 29197.44} C_VEL
LIN {X 0,Y 608.074,Z 1119.047,A -85,B 0,C 180,E1 29195.022,E2 29195.022} C_VEL
LIN {X 0,Y 607.928,Z 1124.49,A -85,B 0,C 180,E1 29192.638,E2 29192.638} C_VEL
LIN {X 0,Y 607.925,Z 1128.438,A -85,B 0,C 180,E1 29190.219,E2 29190.219} C_VEL
LIN {X 0,Y 607.911,Z 1130.882,A -85,B 0,C 180,E1 29187.848,E2 29187.848} C_VEL
LIN {X 0,Y 607.901,Z 1131.894,A -85,B 0,C 180,E1 29185.528,E2 29185.528} C_VEL
LIN {X 0,Y 607.869,Z 1131.51,A -85,B 0,C 180,E1 29183.047,E2 29183.047} C_VEL
LIN {X 0,Y 607.918,Z 1129.587,A -85,B 0,C 180,E1 29180.609,E2 29180.609} C_VEL
LIN {X 0,Y 607.943,Z 1126.184,A -85,B 0,C 180,E1 29178.21,E2 29178.21} C_VEL
LIN {X 0,Y 608.024,Z 1120.952,A -85,B 0,C 180,E1 29175.646,E2 29175.646} C_VEL
LIN {X 0,Y 608.221,Z 1113.755,A -85,B 0,C 180,E1 29173.016,E2 29173.016} C_VEL
LIN {X 0,Y 608.518,Z 1106.224,A -85,B 0,C 180,E1 29170.796,E2 29170.796} C_VEL
LIN {X 0,Y 609.01,Z 1096.673,A -85,B 0,C 180,E1 29168.402,E2 29168.402} C_VEL
LIN {X 0,Y 609.789,Z 1084.508,A -85,B 0,C 180,E1 29165.835,E2 29165.835} C_VEL
LIN {X 0,Y 610.757,Z 1072.024,A -85,B 0,C 180,E1 29163.567,E2 29163.567} C_VEL
LIN {X 0,Y 612.115,Z 1056.683,A -85,B 0,C 180,E1 29161.123,E2 29161.123} C_VEL
LIN {X 0,Y 613.789,Z 1039.863,A -85,B 0,C 180,E1 29158.787,E2 29158.787} C_VEL
LIN {X 0,Y 615.566,Z 1023.277,A -85,B 0,C 180,E1 29156.741,E2 29156.741} C_VEL
LIN {X 0,Y 617.819,Z 1003.765,A -85,B 0,C 180,E1 29154.614,E2 29154.614} C_VEL
LIN {X 0,Y 620.235,Z 983.172,A -85,B 0,C 180,E1 29152.637,E2 29152.637} C_VEL
LIN {X 0,Y 622.997,Z 960.449,A -85,B 0,C 180,E1 29150.718,E2 29150.718} C_VEL
LIN {X 0,Y 625.64,Z 938.427,A -85,B 0,C 180,E1 29149.083,E2 29149.083} C_VEL
LIN {X 0,Y 628.36,Z 914.733,A -85,B 0,C 180,E1 29147.548,E2 29147.548} C_VEL
LIN {X 0,Y 630.984,Z 890.686,A -85,B 0,C 180,E1 29146.202,E2 29146.202} C_VEL
LIN {X 0,Y 633.558,Z 865.629,A -85,B 0,C 180,E1 29144.999,E2 29144.999} C_VEL
LIN {X 0,Y 635.849,Z 840.553,A -85,B 0,C 180,E1 29143.98,E2 29143.98} C_VEL
LIN {X 0,Y 637.875,Z 814.71,A -85,B 0,C 180,E1 29143.119,E2 29143.119} C_VEL
LIN {X 0,Y 639.668,Z 788.289,A -85,B 0,C 180,E1 29142.415,E2 29142.415} C_VEL
LIN {X 0,Y 640.966,Z 763.391,A -85,B 0,C 180,E1 29141.912,E2 29141.912} C_VEL
LIN {X 0,Y 642.06,Z 726.634,A -85,B 0,C 180,E1 29141.378,E2 29141.378} C_VEL
LIN {X 0,Y 644.87,Z 581.78,A -85,B 0,C 180,E1 29139.448,E2 29139.448} C_VEL
LIN {X 0,Y 647.968,Z 422.761,A -85,B 0,C 180,E1 29137.303,E2 29137.303} C_VEL
LIN {X 0,Y 648.369,Z 399.781,A -85,B 0,C 180,E1 29136.966,E2 29136.966} C_VEL
LIN {X 0,Y 635.235,Z 381.178,A -85,B 0,C 180,E1 29135.313,E2 29135.313} C_VEL
LIN {X 0,Y 628.974,Z 372.167,A -85,B 0,C 180,E1 29134.38,E2 29134.38} C_VEL
LIN {X 0,Y 625.668,Z 367.465,A -85,B 0,C 180,E1 29133.819,E2 29133.819} C_VEL
LIN {X 0,Y 622.516,Z 363.133,A -85,B 0,C 180,E1 29133.257,E2 29133.257} C_VEL
LIN {X 0,Y 619.539,Z 359.232,A -85,B 0,C 180,E1 29132.654,E2 29132.654} C_VEL
LIN {X 0,Y 618.634,Z 357.785,A -85,B 0,C 180,E1 29132.449,E2 29132.449} C_VEL
LIN {X 0,Y 615.699,Z 354.813,A -85,B 0,C 180,E1 29131.763,E2 29131.763} C_VEL
LIN {X 0,Y 614.205,Z 351.973,A -85,B 0,C 180,E1 29131.299,E2 29131.299} C_VEL
LIN {X 0,Y 610.868,Z 349.488,A -85,B 0,C 180,E1 29130.11,E2 29130.11} C_VEL
LIN {X 0,Y 609.559,Z 347.366,A -85,B 0,C 180,E1 29129.08,E2 29129.08} C_VEL
LIN {X 0,Y 609.711,Z 347.673,A -85,B 0,C 180,E1 29128.787,E2 29128.787} C_VEL
LIN {X 0,Y 611.757,Z 350.678,A -85,B 0,C 180,E1 29127.803,E2 29127.803} C_VEL
LIN {X 0,Y 613.456,Z 354.356,A -85,B 0,C 180,E1 29127.016,E2 29127.016} C_VEL
LIN {X 0,Y 614.677,Z 356.97,A -85,B 0,C 180,E1 29126.533,E2 29126.533} C_VEL
LIN {X 0,Y 616.59,Z 360.935,A -85,B 0,C 180,E1 29125.869,E2 29125.869} C_VEL
LIN {X 0,Y 620.519,Z 369.593,A -85,B 0,C 180,E1 29124.656,E2 29124.656} C_VEL
LIN {X 0,Y 625.498,Z 382.519,A -85,B 0,C 180,E1 29123.212,E2 29123.212} C_VEL
LIN {X 0,Y 631.076,Z 396.665,A -85,B 0,C 180,E1 29121.835,E2 29121.835} C_VEL
LIN {X 0,Y 637.33,Z 406.869,A -85,B 0,C 180,E1 29120.964,E2 29120.964} C_VEL
LIN {X 0,Y 644.468,Z 447.377,A -85,B 0,C 180,E1 29119.598,E2 29119.598} C_VEL
LIN {X 0,Y 648.435,Z 465.96,A -85,B 0,C 180,E1 29118.967,E2 29118.967} C_VEL
LIN {X 0,Y 645.891,Z 635.975,A -85,B 0,C 180,E1 29116.707,E2 29116.707} C_VEL
LIN {X 0,Y 643.983,Z 784.635,A -85,B 0,C 180,E1 29114.814,E2 29114.814} C_VEL
LIN {X 0,Y 641.298,Z 904.689,A -85,B 0,C 180,E1 29113.184,E2 29113.184} C_VEL
LIN {X 0,Y 640.081,Z 931.504,A -85,B 0,C 180,E1 29112.695,E2 29112.695} C_VEL
LIN {X 0,Y 638.344,Z 958.109,A -85,B 0,C 180,E1 29112.026,E2 29112.026} C_VEL
LIN {X 0,Y 636.7,Z 979.746,A -85,B 0,C 180,E1 29111.352,E2 29111.352} C_VEL
LIN {X 0,Y 634.94,Z 1000.2,A -85,B 0,C 180,E1 29110.6,E2 29110.6} C_VEL
LIN {X 0,Y 632.779,Z 1023.23,A -85,B 0,C 180,E1 29109.612,E2 29109.612} C_VEL
LIN {X 0,Y 630.083,Z 1049.23,A -85,B 0,C 180,E1 29108.293,E2 29108.293} C_VEL
LIN {X 0,Y 627.84,Z 1069.186,A -85,B 0,C 180,E1 29107.127,E2 29107.127} C_VEL
LIN {X 0,Y 625.613,Z 1088.303,A -85,B 0,C 180,E1 29105.873,E2 29105.873} C_VEL
LIN {X 0,Y 623.339,Z 1107.548,A -85,B 0,C 180,E1 29104.462,E2 29104.462} C_VEL
LIN {X 0,Y 620.566,Z 1130.5,A -85,B 0,C 180,E1 29102.558,E2 29102.558} C_VEL
LIN {X 0,Y 618.367,Z 1148.78,A -85,B 0,C 180,E1 29100.836,E2 29100.836} C_VEL
LIN {X 0,Y 616.508,Z 1164.765,A -85,B 0,C 180,E1 29099.167,E2 29099.167} C_VEL
LIN {X 0,Y 614.574,Z 1182.598,A -85,B 0,C 180,E1 29097.1,E2 29097.1} C_VEL
LIN {X 0,Y 612.753,Z 1199.988,A -85,B 0,C 180,E1 29094.795,E2 29094.795} C_VEL
LIN {X 0,Y 611.454,Z 1213.787,A -85,B 0,C 180,E1 29092.736,E2 29092.736} C_VEL
LIN {X 0,Y 610.225,Z 1228.628,A -85,B 0,C 180,E1 29090.226,E2 29090.226} C_VEL
LIN {X 0,Y 609.356,Z 1240.616,A -85,B 0,C 180,E1 29087.869,E2 29087.869} C_VEL
LIN {X 0,Y 608.805,Z 1249.992,A -85,B 0,C 180,E1 29085.753,E2 29085.753} C_VEL
LIN {X 0,Y 608.39,Z 1258.633,A -85,B 0,C 180,E1 29083.496,E2 29083.496} C_VEL
LIN {X 0,Y 608.117,Z 1266.777,A -85,B 0,C 180,E1 29080.899,E2 29080.899} C_VEL
LIN {X 0,Y 608.004,Z 1272.728,A -85,B 0,C 180,E1 29078.511,E2 29078.511} C_VEL
LIN {X 0,Y 607.936,Z 1277.337,A -85,B 0,C 180,E1 29076.042,E2 29076.042} C_VEL
LIN {X 0,Y 607.912,Z 1280.404,A -85,B 0,C 180,E1 29073.489,E2 29073.489} C_VEL
LIN {X 0,Y 607.891,Z 1281.714,A -85,B 0,C 180,E1 29071.225,E2 29071.225} C_VEL
LIN {X 0,Y 607.864,Z 1281.827,A -85,B 0,C 180,E1 29069.246,E2 29069.246} C_VEL
LIN {X 0,Y 607.909,Z 1280.947,A -85,B 0,C 180,E1 29067.266,E2 29067.266} C_VEL
LIN {X 0,Y 607.917,Z 1279.006,A -85,B 0,C 180,E1 29065.188,E2 29065.188} C_VEL
LIN {X 0,Y 607.958,Z 1275.422,A -85,B 0,C 180,E1 29062.82,E2 29062.82} C_VEL
LIN {X 0,Y 608.01,Z 1270.091,A -85,B 0,C 180,E1 29060.344,E2 29060.344} C_VEL
LIN {X 0,Y 608.215,Z 1263.534,A -85,B 0,C 180,E1 29058.006,E2 29058.006} C_VEL
LIN {X 0,Y 608.442,Z 1256.865,A -85,B 0,C 180,E1 29056.021,E2 29056.021} C_VEL
LIN {X 0,Y 608.874,Z 1248.901,A -85,B 0,C 180,E1 29053.985,E2 29053.985} C_VEL
LIN {X 0,Y 609.449,Z 1239.02,A -85,B 0,C 180,E1 29051.794,E2 29051.794} C_VEL
LIN {X 0,Y 610.427,Z 1225.869,A -85,B 0,C 180,E1 29049.279,E2 29049.279} C_VEL
LIN {X 0,Y 611.545,Z 1212.739,A -85,B 0,C 180,E1 29047.1,E2 29047.1} C_VEL
LIN {X 0,Y 612.819,Z 1199.282,A -85,B 0,C 180,E1 29045.105,E2 29045.105} C_VEL
LIN {X 0,Y 614.664,Z 1181.754,A -85,B 0,C 180,E1 29042.8,E2 29042.8} C_VEL
LIN {X 0,Y 616.557,Z 1164.301,A -85,B 0,C 180,E1 29040.782,E2 29040.782} C_VEL
LIN {X 0,Y 618.418,Z 1148.322,A -85,B 0,C 180,E1 29039.119,E2 29039.119} C_VEL
LIN {X 0,Y 620.922,Z 1127.858,A -85,B 0,C 180,E1 29037.203,E2 29037.203} C_VEL
LIN {X 0,Y 623.448,Z 1106.559,A -85,B 0,C 180,E1 29035.463,E2 29035.463} C_VEL
LIN {X 0,Y 625.672,Z 1087.778,A -85,B 0,C 180,E1 29034.091,E2 29034.091} C_VEL
LIN {X 0,Y 627.932,Z 1068.368,A -85,B 0,C 180,E1 29032.822,E2 29032.822} C_VEL
LIN {X 0,Y 630.673,Z 1043.837,A -85,B 0,C 180,E1 29031.409,E2 29031.409} C_VEL
LIN {X 0,Y 633.094,Z 1019.844,A -85,B 0,C 180,E1 29030.235,E2 29030.235} C_VEL
LIN {X 0,Y 634.994,Z 999.56,A -85,B 0,C 180,E1 29029.375,E2 29029.375} C_VEL
LIN {X 0,Y 636.765,Z 978.882,A -85,B 0,C 180,E1 29028.618,E2 29028.618} C_VEL
LIN {X 0,Y 638.512,Z 955.833,A -85,B 0,C 180,E1 29027.908,E2 29027.908} C_VEL
LIN {X 0,Y 640.271,Z 927.304,A -85,B 0,C 180,E1 29027.221,E2 29027.221} C_VEL
LIN {X 0,Y 641.344,Z 903.414,A -85,B 0,C 180,E1 29026.797,E2 29026.797} C_VEL
LIN {X 0,Y 644.774,Z 742.312,A -85,B 0,C 180,E1 29024.624,E2 29024.624} C_VEL
LIN {X 0,Y 648.915,Z 541.096,A -85,B 0,C 180,E1 29021.886,E2 29021.886} C_VEL
LIN {X 0,Y 650.406,Z 464.918,A -85,B 0,C 180,E1 29020.814,E2 29020.814} C_VEL
LIN {X 0,Y 642.032,Z 421.807,A -85,B 0,C 180,E1 29019.183,E2 29019.183} C_VEL
LIN {X 0,Y 642.606,Z 410.822,A -85,B 0,C 180,E1 29018.435,E2 29018.435} C_VEL
LIN {X 0,Y 630.93,Z 386.875,A -85,B 0,C 180,E1 29015.342,E2 29015.342} C_VEL
LIN {X 0,Y 621.864,Z 369.282,A -85,B 0,C 180,E1 29012.81,E2 29012.81} C_VEL
LIN {X 0,Y 616.106,Z 358.958,A -85,B 0,C 180,E1 29011.179,E2 29011.179} C_VEL
LIN {X 0,Y 613.642,Z 354.459,A -85,B 0,C 180,E1 29010.448,E2 29010.448} C_VEL
LIN {X 0,Y 611.139,Z 349.828,A -85,B 0,C 180,E1 29009.685,E2 29009.685} C_VEL
LIN {X 0,Y 609.4,Z 346.822,A -85,B 0,C 180,E1 29009.164,E2 29009.164} C_VEL
LIN {X 0,Y 609.091,Z 345.534,A -85,B 0,C 180,E1 29008.915,E2 29008.915} C_VEL
LIN {X 0,Y 609.07,Z 345.355,A -85,B 0,C 180,E1 29005.676,E2 29005.676} C_VEL
LIN {X 0,Y 609.05,Z 345.368,A -85,B 0,C 180,E1 29002.441,E2 29002.441} C_VEL
LIN {X 0,Y 609.068,Z 345.365,A -85,B 0,C 180,E1 28999.267,E2 28999.267} C_VEL
LIN {X 0,Y 609.046,Z 345.361,A -85,B 0,C 180,E1 28996.108,E2 28996.108} C_VEL
LIN {X 0,Y 609.071,Z 345.362,A -85,B 0,C 180,E1 28992.998,E2 28992.998} C_VEL
LIN {X 0,Y 609.045,Z 345.362,A -85,B 0,C 180,E1 28989.831,E2 28989.831} C_VEL
LIN {X 0,Y 609.075,Z 345.364,A -85,B 0,C 180,E1 28986.599,E2 28986.599} C_VEL
LIN {X 0,Y 609.052,Z 345.362,A -85,B 0,C 180,E1 28983.388,E2 28983.388} C_VEL
LIN {X 0,Y 609.06,Z 345.367,A -85,B 0,C 180,E1 28980.094,E2 28980.094} C_VEL
LIN {X 0,Y 609.069,Z 345.358,A -85,B 0,C 180,E1 28976.894,E2 28976.894} C_VEL
LIN {X 0,Y 609.041,Z 345.363,A -85,B 0,C 180,E1 28973.685,E2 28973.685} C_VEL
LIN {X 0,Y 609.075,Z 345.358,A -85,B 0,C 180,E1 28970.551,E2 28970.551} C_VEL
LIN {X 0,Y 609.035,Z 345.364,A -85,B 0,C 180,E1 28967.388,E2 28967.388} C_VEL
LIN {X 0,Y 609.078,Z 345.36,A -85,B 0,C 180,E1 28964.284,E2 28964.284} C_VEL
LIN {X 0,Y 609.031,Z 345.364,A -85,B 0,C 180,E1 28961.129,E2 28961.129} C_VEL
LIN {X 0,Y 609.078,Z 345.362,A -85,B 0,C 180,E1 28958.019,E2 28958.019} C_VEL
LIN {X 0,Y 609.028,Z 345.364,A -85,B 0,C 180,E1 28954.939,E2 28954.939} C_VEL
LIN {X 0,Y 609.08,Z 345.362,A -85,B 0,C 180,E1 28951.784,E2 28951.784} C_VEL
LIN {X 0,Y 609.025,Z 345.365,A -85,B 0,C 180,E1 28948.748,E2 28948.748} C_VEL
LIN {X 0,Y 609.079,Z 345.362,A -85,B 0,C 180,E1 28945.617,E2 28945.617} C_VEL
LIN {X 0,Y 609.022,Z 345.365,A -85,B 0,C 180,E1 28942.464,E2 28942.464} C_VEL
LIN {X 0,Y 609.082,Z 345.361,A -85,B 0,C 180,E1 28939.451,E2 28939.451} C_VEL
LIN {X 0,Y 609.019,Z 345.366,A -85,B 0,C 180,E1 28936.388,E2 28936.388} C_VEL
LIN {X 0,Y 609.078,Z 345.36,A -85,B 0,C 180,E1 28933.33,E2 28933.33} C_VEL
LIN {X 0,Y 609.015,Z 345.367,A -85,B 0,C 180,E1 28930.231,E2 28930.231} C_VEL
LIN {X 0,Y 609.069,Z 345.36,A -85,B 0,C 180,E1 28927.23,E2 28927.23} C_VEL
LIN {X 0,Y 609.012,Z 345.367,A -85,B 0,C 180,E1 28924.046,E2 28924.046} C_VEL
LIN {X 0,Y 609.014,Z 345.362,A -85,B 0,C 180,E1 28921.661,E2 28921.661} C_VEL
LIN {X 0,Y 608.056,Z 345.489,A -85,B 0,C 180,E1 28920.937,E2 28920.937} C_VEL
LIN {X 0,Y 601.577,Z 346.288,A -85,B 0,C 180,E1 28918.851,E2 28918.851} C_VEL
LIN {X 0,Y 601.105,Z 346.354,A -85,B 0,C 180,E1 28918.375,E2 28918.375} C_VEL
LIN {X 0,Y 601.076,Z 346.351,A -85,B 0,C 180,E1 28915.407,E2 28915.407} C_VEL
LIN {X 0,Y 601.101,Z 346.356,A -85,B 0,C 180,E1 28912.185,E2 28912.185} C_VEL
LIN {X 0,Y 601.066,Z 346.356,A -85,B 0,C 180,E1 28909.332,E2 28909.332} C_VEL
LIN {X 0,Y 601.126,Z 346.354,A -85,B 0,C 180,E1 28906.227,E2 28906.227} C_VEL
LIN {X 0,Y 601.059,Z 346.356,A -85,B 0,C 180,E1 28903.272,E2 28903.272} C_VEL
LIN {X 0,Y 601.129,Z 346.347,A -85,B 0,C 180,E1 28900.155,E2 28900.155} C_VEL
LIN {X 0,Y 601.055,Z 346.354,A -85,B 0,C 180,E1 28897.167,E2 28897.167} C_VEL
LIN {X 0,Y 601.115,Z 346.349,A -85,B 0,C 180,E1 28894.197,E2 28894.197} C_VEL
LIN {X 0,Y 601.052,Z 346.359,A -85,B 0,C 180,E1 28891.049,E2 28891.049} C_VEL
LIN {X 0,Y 601.078,Z 346.343,A -85,B 0,C 180,E1 28888.284,E2 28888.284} C_VEL
LIN {X 0,Y 601.056,Z 346.363,A -85,B 0,C 180,E1 28885.038,E2 28885.038} C_VEL
LIN {X 0,Y 601.06,Z 346.333,A -85,B 0,C 180,E1 28882.256,E2 28882.256} C_VEL
LIN {X 0,Y 601.149,Z 346.54,A -85,B 0,C 180,E1 28879.555,E2 28879.555} C_VEL
LIN {X 0,Y 601.491,Z 347.998,A -85,B 0,C 180,E1 28879.343,E2 28879.343} C_VEL
LIN {X 0,Y 603.314,Z 350.967,A -85,B 0,C 180,E1 28879.037,E2 28879.037} C_VEL
LIN {X 0,Y 605.495,Z 352.918,A -85,B 0,C 180,E1 28878.715,E2 28878.715} C_VEL
LIN {X 0,Y 607.934,Z 356.671,A -85,B 0,C 180,E1 28878.329,E2 28878.329} C_VEL
LIN {X 0,Y 610.04,Z 358.846,A -85,B 0,C 180,E1 28878.022,E2 28878.022} C_VEL
LIN {X 0,Y 613.259,Z 363.12,A -85,B 0,C 180,E1 28877.544,E2 28877.544} C_VEL
LIN {X 0,Y 622.536,Z 375.004,A -85,B 0,C 180,E1 28876.225,E2 28876.225} C_VEL
LIN {X 0,Y 634.063,Z 390.707,A -85,B 0,C 180,E1 28874.661,E2 28874.661} C_VEL
LIN {X 0,Y 643.661,Z 404.186,A -85,B 0,C 180,E1 28873.45,E2 28873.45} C_VEL
LIN {X 0,Y 638.49,Z 619.711,A -85,B 0,C 180,E1 28870.466,E2 28870.466} C_VEL
LIN {X 0,Y 635.462,Z 756.173,A -85,B 0,C 180,E1 28868.616,E2 28868.616} C_VEL
LIN {X 0,Y 634.08,Z 782.508,A -85,B 0,C 180,E1 28868.119,E2 28868.119} C_VEL
LIN {X 0,Y 632.263,Z 809.683,A -85,B 0,C 180,E1 28867.429,E2 28867.429} C_VEL
LIN {X 0,Y 630.274,Z 834.551,A -85,B 0,C 180,E1 28866.634,E2 28866.634} C_VEL
LIN {X 0,Y 627.966,Z 859.2,A -85,B 0,C 180,E1 28865.67,E2 28865.67} C_VEL
LIN {X 0,Y 625.37,Z 883.867,A -85,B 0,C 180,E1 28864.527,E2 28864.527} C_VEL
LIN {X 0,Y 622.769,Z 906.964,A -85,B 0,C 180,E1 28863.285,E2 28863.285} C_VEL
LIN {X 0,Y 619.832,Z 930.889,A -85,B 0,C 180,E1 28861.794,E2 28861.794} C_VEL
LIN {X 0,Y 616.891,Z 954.044,A -85,B 0,C 180,E1 28860.13,E2 28860.13} C_VEL
LIN {X 0,Y 614.108,Z 976.086,A -85,B 0,C 180,E1 28858.326,E2 28858.326} C_VEL
LIN {X 0,Y 611.398,Z 997.313,A -85,B 0,C 180,E1 28856.349,E2 28856.349} C_VEL
LIN {X 0,Y 609.029,Z 1016.213,A -85,B 0,C 180,E1 28854.351,E2 28854.351} C_VEL
LIN {X 0,Y 606.775,Z 1035.252,A -85,B 0,C 180,E1 28852.074,E2 28852.074} C_VEL
LIN {X 0,Y 604.906,Z 1052.431,A -85,B 0,C 180,E1 28849.737,E2 28849.737} C_VEL
LIN {X 0,Y 603.3,Z 1068.461,A -85,B 0,C 180,E1 28847.241,E2 28847.241} C_VEL
LIN {X 0,Y 602.192,Z 1081.139,A -85,B 0,C 180,E1 28844.982,E2 28844.982} C_VEL
LIN {X 0,Y 601.336,Z 1093.003,A -85,B 0,C 180,E1 28842.557,E2 28842.557} C_VEL
LIN {X 0,Y 600.679,Z 1103.743,A -85,B 0,C 180,E1 28839.981,E2 28839.981} C_VEL
LIN {X 0,Y 600.296,Z 1111.791,A -85,B 0,C 180,E1 28837.684,E2 28837.684} C_VEL
LIN {X 0,Y 600.086,Z 1118.922,A -85,B 0,C 180,E1 28835.206,E2 28835.206} C_VEL
LIN {X 0,Y 599.93,Z 1124.374,A -85,B 0,C 180,E1 28832.798,E2 28832.798} C_VEL
LIN {X 0,Y 599.926,Z 1128.232,A -85,B 0,C 180,E1 28830.443,E2 28830.443} C_VEL
LIN {X 0,Y 599.918,Z 1130.779,A -85,B 0,C 180,E1 28828.035,E2 28828.035} C_VEL
LIN {X 0,Y 599.906,Z 1131.866,A -85,B 0,C 180,E1 28825.681,E2 28825.681} C_VEL
LIN {X 0,Y 599.883,Z 1131.644,A -85,B 0,C 180,E1 28823.268,E2 28823.268} C_VEL
LIN {X 0,Y 599.918,Z 1129.738,A -85,B 0,C 180,E1 28820.692,E2 28820.692} C_VEL
LIN {X 0,Y 599.945,Z 1126.25,A -85,B 0,C 180,E1 28818.159,E2 28818.159} C_VEL
LIN {X 0,Y 600.035,Z 1121.052,A -85,B 0,C 180,E1 28815.563,E2 28815.563} C_VEL
LIN {X 0,Y 600.236,Z 1113.895,A -85,B 0,C 180,E1 28812.898,E2 28812.898} C_VEL
LIN {X 0,Y 600.586,Z 1106.033,A -85,B 0,C 180,E1 28810.552,E2 28810.552} C_VEL
LIN {X 0,Y 601.131,Z 1096.035,A -85,B 0,C 180,E1 28808.032,E2 28808.032} C_VEL
LIN {X 0,Y 601.994,Z 1083.76,A -85,B 0,C 180,E1 28805.433,E2 28805.433} C_VEL
LIN {X 0,Y 603.063,Z 1071.209,A -85,B 0,C 180,E1 28803.137,E2 28803.137} C_VEL
LIN {X 0,Y 604.495,Z 1056.386,A -85,B 0,C 180,E1 28800.758,E2 28800.758} C_VEL
LIN {X 0,Y 606.292,Z 1039.537,A -85,B 0,C 180,E1 28798.393,E2 28798.393} C_VEL
LIN {X 0,Y 608.234,Z 1022.918,A -85,B 0,C 180,E1 28796.324,E2 28796.324} C_VEL
LIN {X 0,Y 610.741,Z 1002.475,A -85,B 0,C 180,E1 28794.08,E2 28794.08} C_VEL
LIN {X 0,Y 613.295,Z 982.193,A -85,B 0,C 180,E1 28792.129,E2 28792.129} C_VEL
LIN {X 0,Y 616.182,Z 959.891,A -85,B 0,C 180,E1 28790.237,E2 28790.237} C_VEL
LIN {X 0,Y 618.985,Z 937.805,A -85,B 0,C 180,E1 28788.587,E2 28788.587} C_VEL
LIN {X 0,Y 621.99,Z 913.264,A -85,B 0,C 180,E1 28786.994,E2 28786.994} C_VEL
LIN {X 0,Y 624.704,Z 889.768,A -85,B 0,C 180,E1 28785.683,E2 28785.683} C_VEL
LIN {X 0,Y 627.319,Z 865.523,A -85,B 0,C 180,E1 28784.515,E2 28784.515} C_VEL
LIN {X 0,Y 629.621,Z 841.558,A -85,B 0,C 180,E1 28783.532,E2 28783.532} C_VEL
LIN {X 0,Y 631.794,Z 815.561,A -85,B 0,C 180,E1 28782.655,E2 28782.655} C_VEL
LIN {X 0,Y 633.673,Z 789.621,A -85,B 0,C 180,E1 28781.952,E2 28781.952} C_VEL
LIN {X 0,Y 635.063,Z 764.375,A -85,B 0,C 180,E1 28781.434,E2 28781.434} C_VEL
LIN {X 0,Y 636.229,Z 728.301,A -85,B 0,C 180,E1 28780.902,E2 28780.902} C_VEL
LIN {X 0,Y 640.094,Z 516.168,A -85,B 0,C 180,E1 28778.097,E2 28778.097} C_VEL
LIN {X 0,Y 642.836,Z 403.816,A -85,B 0,C 180,E1 28776.515,E2 28776.515} C_VEL
LIN {X 0,Y 629.876,Z 384.93,A -85,B 0,C 180,E1 28774.77,E2 28774.77} C_VEL
LIN {X 0,Y 624.871,Z 377.684,A -85,B 0,C 180,E1 28773.968,E2 28773.968} C_VEL
LIN {X 0,Y 621.923,Z 373.489,A -85,B 0,C 180,E1 28773.452,E2 28773.452} C_VEL
LIN {X 0,Y 619.531,Z 370.015,A -85,B 0,C 180,E1 28772.985,E2 28772.985} C_VEL
LIN {X 0,Y 616.485,Z 365.687,A -85,B 0,C 180,E1 28772.32,E2 28772.32} C_VEL
LIN {X 0,Y 612.885,Z 361.273,A -85,B 0,C 180,E1 28771.396,E2 28771.396} C_VEL
LIN {X 0,Y 611.993,Z 359.473,A -85,B 0,C 180,E1 28771.078,E2 28771.078} C_VEL
LIN {X 0,Y 609.02,Z 357.018,A -85,B 0,C 180,E1 28769.907,E2 28769.907} C_VEL
LIN {X 0,Y 607.994,Z 355.266,A -85,B 0,C 180,E1 28768.96,E2 28768.96} C_VEL
LIN {X 0,Y 607.622,Z 357.674,A -85,B 0,C 180,E1 28767.891,E2 28767.891} C_VEL
LIN {X 0,Y 608.475,Z 360.626,A -85,B 0,C 180,E1 28767.049,E2 28767.049} C_VEL
LIN {X 0,Y 611.168,Z 366.744,A -85,B 0,C 180,E1 28765.977,E2 28765.977} C_VEL
LIN {X 0,Y 614.918,Z 375.427,A -85,B 0,C 180,E1 28764.742,E2 28764.742} C_VEL
LIN {X 0,Y 618.337,Z 384.101,A -85,B 0,C 180,E1 28763.755,E2 28763.755} C_VEL
LIN {X 0,Y 626.224,Z 401.248,A -85,B 0,C 180,E1 28762.27,E2 28762.27} C_VEL
LIN {X 0,Y 632.423,Z 411.695,A -85,B 0,C 180,E1 28761.368,E2 28761.368} C_VEL
LIN {X 0,Y 638.881,Z 450.544,A -85,B 0,C 180,E1 28760.024,E2 28760.024} C_VEL
LIN {X 0,Y 642.52,Z 467.863,A -85,B 0,C 180,E1 28759.427,E2 28759.427} C_VEL
LIN {X 0,Y 639.982,Z 606.569,A -85,B 0,C 180,E1 28757.531,E2 28757.531} C_VEL
LIN {X 0,Y 637.279,Z 812.128,A -85,B 0,C 180,E1 28754.907,E2 28754.907} C_VEL
LIN {X 0,Y 635.854,Z 894.278,A -85,B 0,C 180,E1 28753.835,E2 28753.835} C_VEL
LIN {X 0,Y 634.762,Z 919.756,A -85,B 0,C 180,E1 28753.421,E2 28753.421} C_VEL
LIN {X 0,Y 633.495,Z 941.481,A -85,B 0,C 180,E1 28752.953,E2 28752.953} C_VEL
LIN {X 0,Y 631.974,Z 963.094,A -85,B 0,C 180,E1 28752.372,E2 28752.372} C_VEL
LIN {X 0,Y 629.964,Z 987.758,A -85,B 0,C 180,E1 28751.563,E2 28751.563} C_VEL
LIN {X 0,Y 627.435,Z 1014.185,A -85,B 0,C 180,E1 28750.495,E2 28750.495} C_VEL
LIN {X 0,Y 625.261,Z 1034.673,A -85,B 0,C 180,E1 28749.528,E2 28749.528} C_VEL
LIN {X 0,Y 623.097,Z 1053.728,A -85,B 0,C 180,E1 28748.508,E2 28748.508} C_VEL
LIN {X 0,Y 620.861,Z 1072.428,A -85,B 0,C 180,E1 28747.383,E2 28747.383} C_VEL
LIN {X 0,Y 618.338,Z 1092.926,A -85,B 0,C 180,E1 28746,E2 28746} C_VEL
LIN {X 0,Y 615.313,Z 1116.359,A -85,B 0,C 180,E1 28744.195,E2 28744.195} C_VEL
LIN {X 0,Y 612.994,Z 1134.383,A -85,B 0,C 180,E1 28742.622,E2 28742.622} C_VEL
LIN {X 0,Y 610.877,Z 1151.132,A -85,B 0,C 180,E1 28741.001,E2 28741.001} C_VEL
LIN {X 0,Y 608.621,Z 1169.853,A -85,B 0,C 180,E1 28738.989,E2 28738.989} C_VEL
LIN {X 0,Y 606.423,Z 1188.075,A -85,B 0,C 180,E1 28736.752,E2 28736.752} C_VEL
LIN {X 0,Y 604.929,Z 1202.086,A -85,B 0,C 180,E1 28734.824,E2 28734.824} C_VEL
LIN {X 0,Y 603.451,Z 1217.179,A -85,B 0,C 180,E1 28732.504,E2 28732.504} C_VEL
LIN {X 0,Y 602.204,Z 1231.324,A -85,B 0,C 180,E1 28729.985,E2 28729.985} C_VEL
LIN {X 0,Y 601.396,Z 1241.99,A -85,B 0,C 180,E1 28727.813,E2 28727.813} C_VEL
LIN {X 0,Y 600.748,Z 1252.943,A -85,B 0,C 180,E1 28725.246,E2 28725.246} C_VEL
LIN {X 0,Y 600.318,Z 1261.836,A -85,B 0,C 180,E1 28722.701,E2 28722.701} C_VEL
LIN {X 0,Y 600.112,Z 1268.057,A -85,B 0,C 180,E1 28720.561,E2 28720.561} C_VEL
LIN {X 0,Y 599.993,Z 1273.344,A -85,B 0,C 180,E1 28718.336,E2 28718.336} C_VEL
LIN {X 0,Y 599.934,Z 1277.782,A -85,B 0,C 180,E1 28715.835,E2 28715.835} C_VEL
LIN {X 0,Y 599.91,Z 1280.54,A -85,B 0,C 180,E1 28713.344,E2 28713.344} C_VEL
LIN {X 0,Y 599.892,Z 1281.714,A -85,B 0,C 180,E1 28711.242,E2 28711.242} C_VEL
LIN {X 0,Y 599.864,Z 1281.827,A -85,B 0,C 180,E1 28709.236,E2 28709.236} C_VEL
LIN {X 0,Y 599.908,Z 1281.015,A -85,B 0,C 180,E1 28707.325,E2 28707.325} C_VEL
LIN {X 0,Y 599.916,Z 1279.117,A -85,B 0,C 180,E1 28705.22,E2 28705.22} C_VEL
LIN {X 0,Y 599.959,Z 1275.59,A -85,B 0,C 180,E1 28702.82,E2 28702.82} C_VEL
LIN {X 0,Y 600.03,Z 1270.091,A -85,B 0,C 180,E1 28700.214,E2 28700.214} C_VEL
LIN {X 0,Y 600.237,Z 1263.657,A -85,B 0,C 180,E1 28697.884,E2 28697.884} C_VEL
LIN {X 0,Y 600.5,Z 1256.864,A -85,B 0,C 180,E1 28695.832,E2 28695.832} C_VEL
LIN {X 0,Y 600.963,Z 1248.9,A -85,B 0,C 180,E1 28693.769,E2 28693.769} C_VEL
LIN {X 0,Y 601.568,Z 1239.225,A -85,B 0,C 180,E1 28691.591,E2 28691.591} C_VEL
LIN {X 0,Y 602.637,Z 1225.873,A -85,B 0,C 180,E1 28688.999,E2 28688.999} C_VEL
LIN {X 0,Y 603.857,Z 1212.667,A -85,B 0,C 180,E1 28686.78,E2 28686.78} C_VEL
LIN {X 0,Y 605.291,Z 1198.573,A -85,B 0,C 180,E1 28684.669,E2 28684.669} C_VEL
LIN {X 0,Y 607.389,Z 1180.061,A -85,B 0,C 180,E1 28682.233,E2 28682.233} C_VEL
LIN {X 0,Y 609.267,Z 1163.975,A -85,B 0,C 180,E1 28680.36,E2 28680.36} C_VEL
LIN {X 0,Y 611.305,Z 1147.764,A -85,B 0,C 180,E1 28678.659,E2 28678.659} C_VEL
LIN {X 0,Y 613.994,Z 1127.108,A -85,B 0,C 180,E1 28676.716,E2 28676.716} C_VEL
LIN {X 0,Y 616.654,Z 1105.877,A -85,B 0,C 180,E1 28674.97,E2 28674.97} C_VEL
LIN {X 0,Y 619.039,Z 1086.967,A -85,B 0,C 180,E1 28673.582,E2 28673.582} C_VEL
LIN {X 0,Y 621.633,Z 1065.93,A -85,B 0,C 180,E1 28672.206,E2 28672.206} C_VEL
LIN {X 0,Y 624.589,Z 1040.707,A -85,B 0,C 180,E1 28670.777,E2 28670.777} C_VEL
LIN {X 0,Y 626.823,Z 1019.841,A -85,B 0,C 180,E1 28669.757,E2 28669.757} C_VEL
LIN {X 0,Y 628.823,Z 999.566,A -85,B 0,C 180,E1 28668.891,E2 28668.891} C_VEL
LIN {X 0,Y 630.689,Z 978.879,A -85,B 0,C 180,E1 28668.13,E2 28668.13} C_VEL
LIN {X 0,Y 632.495,Z 956.229,A -85,B 0,C 180,E1 28667.428,E2 28667.428} C_VEL
LIN {X 0,Y 634.367,Z 927.623,A -85,B 0,C 180,E1 28666.733,E2 28666.733} C_VEL
LIN {X 0,Y 635.501,Z 903.703,A -85,B 0,C 180,E1 28666.306,E2 28666.306} C_VEL
LIN {X 0,Y 637.188,Z 828.602,A -85,B 0,C 180,E1 28665.289,E2 28665.289} C_VEL
LIN {X 0,Y 640.983,Z 646.522,A -85,B 0,C 180,E1 28662.83,E2 28662.83} C_VEL
LIN {X 0,Y 645.076,Z 467.359,A -85,B 0,C 180,E1 28660.327,E2 28660.327} C_VEL
LIN {X 0,Y 636.2,Z 420.9,A -85,B 0,C 180,E1 28658.542,E2 28658.542} C_VEL
LIN {X 0,Y 636.388,Z 415.1,A -85,B 0,C 180,E1 28658.133,E2 28658.133} C_VEL
LIN {X 0,Y 625.354,Z 392.192,A -85,B 0,C 180,E1 28655.143,E2 28655.143} C_VEL
LIN {X 0,Y 616.305,Z 374.686,A -85,B 0,C 180,E1 28652.591,E2 28652.591} C_VEL
LIN {X 0,Y 608.818,Z 360.828,A -85,B 0,C 180,E1 28650.387,E2 28650.387} C_VEL
LIN {X 0,Y 605.737,Z 355.456,A -85,B 0,C 180,E1 28649.466,E2 28649.466} C_VEL
LIN {X 0,Y 603.395,Z 351.04,A -85,B 0,C 180,E1 28648.722,E2 28648.722} C_VEL
LIN {X 0,Y 601.537,Z 348.073,A -85,B 0,C 180,E1 28648.169,E2 28648.169} C_VEL
LIN {X 0,Y 601.159,Z 346.509,A -85,B 0,C 180,E1 28647.864,E2 28647.864} C_VEL
LIN {X 0,Y 601.115,Z 346.348,A -85,B 0,C 180,E1 28644.573,E2 28644.573} C_VEL
LIN {X 0,Y 601.131,Z 346.342,A -85,B 0,C 180,E1 28641.465,E2 28641.465} C_VEL
LIN {X 0,Y 601.109,Z 346.341,A -85,B 0,C 180,E1 28638.324,E2 28638.324} C_VEL
LIN {X 0,Y 601.129,Z 346.339,A -85,B 0,C 180,E1 28635.138,E2 28635.138} C_VEL
LIN {X 0,Y 601.104,Z 346.34,A -85,B 0,C 180,E1 28632.001,E2 28632.001} C_VEL
LIN {X 0,Y 601.132,Z 346.339,A -85,B 0,C 180,E1 28628.802,E2 28628.802} C_VEL
LIN {X 0,Y 601.103,Z 346.342,A -85,B 0,C 180,E1 28625.728,E2 28625.728} C_VEL
LIN {X 0,Y 601.132,Z 346.344,A -85,B 0,C 180,E1 28622.479,E2 28622.479} C_VEL
LIN {X 0,Y 601.107,Z 346.35,A -85,B 0,C 180,E1 28619.333,E2 28619.333} C_VEL
LIN {X 0,Y 601.118,Z 346.354,A -85,B 0,C 180,E1 28615.994,E2 28615.994} C_VEL
LIN {X 0,Y 601.14,Z 346.345,A -85,B 0,C 180,E1 28612.738,E2 28612.738} C_VEL
LIN {X 0,Y 601.097,Z 346.352,A -85,B 0,C 180,E1 28609.457,E2 28609.457} C_VEL
LIN {X 0,Y 601.138,Z 346.349,A -85,B 0,C 180,E1 28606.338,E2 28606.338} C_VEL
LIN {X 0,Y 601.092,Z 346.345,A -85,B 0,C 180,E1 28603.175,E2 28603.175} C_VEL
LIN {X 0,Y 601.139,Z 346.346,A -85,B 0,C 180,E1 28600.012,E2 28600.012} C_VEL
LIN {X 0,Y 601.089,Z 346.344,A -85,B 0,C 180,E1 28596.885,E2 28596.885} C_VEL
LIN {X 0,Y 601.137,Z 346.345,A -85,B 0,C 180,E1 28593.705,E2 28593.705} C_VEL
LIN {X 0,Y 601.088,Z 346.345,A -85,B 0,C 180,E1 28590.612,E2 28590.612} C_VEL
LIN {X 0,Y 601.135,Z 346.346,A -85,B 0,C 180,E1 28587.49,E2 28587.49} C_VEL
LIN {X 0,Y 601.084,Z 346.346,A -85,B 0,C 180,E1 28584.432,E2 28584.432} C_VEL
LIN {X 0,Y 601.141,Z 346.345,A -85,B 0,C 180,E1 28581.268,E2 28581.268} C_VEL
LIN {X 0,Y 601.083,Z 346.347,A -85,B 0,C 180,E1 28578.179,E2 28578.179} C_VEL
LIN {X 0,Y 601.125,Z 346.346,A -85,B 0,C 180,E1 28574.985,E2 28574.985} C_VEL
LIN {X 0,Y 601.08,Z 346.348,A -85,B 0,C 180,E1 28571.962,E2 28571.962} C_VEL
LIN {X 0,Y 601.114,Z 346.347,A -85,B 0,C 180,E1 28568.714,E2 28568.714} C_VEL
LIN {X 0,Y 601.08,Z 346.349,A -85,B 0,C 180,E1 28565.724,E2 28565.724} C_VEL
LIN {X 0,Y 601.105,Z 346.348,A -85,B 0,C 180,E1 28562.498,E2 28562.498} C_VEL
LIN {X 0,Y 601.072,Z 346.348,A -85,B 0,C 180,E1 28559.608,E2 28559.608} C_VEL
LIN {X 0,Y 601.105,Z 346.354,A -85,B 0,C 180,E1 28558.375,E2 28558.375} C_VEL
LIN {X 0,Y 600.059,Z 346.492,A -85,B 0,C 180,E1 28557.641,E2 28557.641} C_VEL
LIN {X 0,Y 593.648,Z 347.277,A -85,B 0,C 180,E1 28555.581,E2 28555.581} C_VEL
LIN {X 0,Y 593.164,Z 347.339,A -85,B 0,C 180,E1 28555.045,E2 28555.045} C_VEL
LIN {X 0,Y 593.135,Z 347.343,A -85,B 0,C 180,E1 28551.873,E2 28551.873} C_VEL
LIN {X 0,Y 593.15,Z 347.344,A -85,B 0,C 180,E1 28548.968,E2 28548.968} C_VEL
LIN {X 0,Y 593.132,Z 347.341,A -85,B 0,C 180,E1 28545.722,E2 28545.722} C_VEL
LIN {X 0,Y 593.131,Z 347.344,A -85,B 0,C 180,E1 28542.956,E2 28542.956} C_VEL
LIN {X 0,Y 593.135,Z 347.342,A -85,B 0,C 180,E1 28539.607,E2 28539.607} C_VEL
LIN {X 0,Y 593.128,Z 347.343,A -85,B 0,C 180,E1 28536.777,E2 28536.777} C_VEL
LIN {X 0,Y 593.136,Z 347.346,A -85,B 0,C 180,E1 28533.479,E2 28533.479} C_VEL
LIN {X 0,Y 593.123,Z 347.343,A -85,B 0,C 180,E1 28530.58,E2 28530.58} C_VEL
LIN {X 0,Y 593.129,Z 347.314,A -85,B 0,C 180,E1 28527.295,E2 28527.295} C_VEL
LIN {X 0,Y 593.12,Z 347.338,A -85,B 0,C 180,E1 28524.389,E2 28524.389} C_VEL
LIN {X 0,Y 593.126,Z 347.352,A -85,B 0,C 180,E1 28521.071,E2 28521.071} C_VEL
LIN {X 0,Y 593.153,Z 347.666,A -85,B 0,C 180,E1 28520.589,E2 28520.589} C_VEL
LIN {X 0,Y 593.654,Z 349.393,A -85,B 0,C 180,E1 28520.365,E2 28520.365} C_VEL
LIN {X 0,Y 595.701,Z 352.261,A -85,B 0,C 180,E1 28520.02,E2 28520.02} C_VEL
LIN {X 0,Y 597.7,Z 353.95,A -85,B 0,C 180,E1 28519.713,E2 28519.713} C_VEL
LIN {X 0,Y 600.086,Z 357.688,A -85,B 0,C 180,E1 28519.315,E2 28519.315} C_VEL
LIN {X 0,Y 602.266,Z 359.986,A -85,B 0,C 180,E1 28518.981,E2 28518.981} C_VEL
LIN {X 0,Y 605.521,Z 364.255,A -85,B 0,C 180,E1 28518.475,E2 28518.475} C_VEL
LIN {X 0,Y 607.476,Z 366.849,A -85,B 0,C 180,E1 28518.175,E2 28518.175} C_VEL
LIN {X 0,Y 611.766,Z 372.307,A -85,B 0,C 180,E1 28517.541,E2 28517.541} C_VEL
LIN {X 0,Y 618.89,Z 381.379,A -85,B 0,C 180,E1 28516.521,E2 28516.521} C_VEL
LIN {X 0,Y 630.355,Z 397.08,A -85,B 0,C 180,E1 28514.945,E2 28514.945} C_VEL
LIN {X 0,Y 638.228,Z 408.223,A -85,B 0,C 180,E1 28513.932,E2 28513.932} C_VEL
LIN {X 0,Y 632.723,Z 620.629,A -85,B 0,C 180,E1 28510.959,E2 28510.959} C_VEL
LIN {X 0,Y 629.49,Z 758.506,A -85,B 0,C 180,E1 28509.074,E2 28509.074} C_VEL
LIN {X 0,Y 628.049,Z 785.098,A -85,B 0,C 180,E1 28508.561,E2 28508.561} C_VEL
LIN {X 0,Y 626.233,Z 810.732,A -85,B 0,C 180,E1 28507.898,E2 28507.898} C_VEL
LIN {X 0,Y 624.107,Z 835.677,A -85,B 0,C 180,E1 28507.089,E2 28507.089} C_VEL
LIN {X 0,Y 621.69,Z 860.23,A -85,B 0,C 180,E1 28506.118,E2 28506.118} C_VEL
LIN {X 0,Y 618.998,Z 884.355,A -85,B 0,C 180,E1 28504.987,E2 28504.987} C_VEL
LIN {X 0,Y 616.186,Z 907.915,A -85,B 0,C 180,E1 28503.705,E2 28503.705} C_VEL
LIN {X 0,Y 613.219,Z 930.838,A -85,B 0,C 180,E1 28502.262,E2 28502.262} C_VEL
LIN {X 0,Y 610.133,Z 953.669,A -85,B 0,C 180,E1 28500.611,E2 28500.611} C_VEL
LIN {X 0,Y 607.206,Z 975.536,A -85,B 0,C 180,E1 28498.81,E2 28498.81} C_VEL
LIN {X 0,Y 604.299,Z 997.03,A -85,B 0,C 180,E1 28496.793,E2 28496.793} C_VEL
LIN {X 0,Y 601.761,Z 1015.798,A -85,B 0,C 180,E1 28494.791,E2 28494.791} C_VEL
LIN {X 0,Y 599.37,Z 1034.853,A -85,B 0,C 180,E1 28492.49,E2 28492.49} C_VEL
LIN {X 0,Y 597.323,Z 1052.091,A -85,B 0,C 180,E1 28490.125,E2 28490.125} C_VEL
LIN {X 0,Y 595.668,Z 1067.621,A -85,B 0,C 180,E1 28487.693,E2 28487.693} C_VEL
LIN {X 0,Y 594.42,Z 1080.802,A -85,B 0,C 180,E1 28485.322,E2 28485.322} C_VEL
LIN {X 0,Y 593.459,Z 1093.148,A -85,B 0,C 180,E1 28482.765,E2 28482.765} C_VEL
LIN {X 0,Y 592.728,Z 1103.983,A -85,B 0,C 180,E1 28480.122,E2 28480.122} C_VEL
LIN {X 0,Y 592.33,Z 1112.003,A -85,B 0,C 180,E1 28477.79,E2 28477.79} C_VEL
LIN {X 0,Y 592.092,Z 1119.087,A -85,B 0,C 180,E1 28475.279,E2 28475.279} C_VEL
LIN {X 0,Y 591.934,Z 1124.511,A -85,B 0,C 180,E1 28472.836,E2 28472.836} C_VEL
LIN {X 0,Y 591.926,Z 1128.32,A -85,B 0,C 180,E1 28470.449,E2 28470.449} C_VEL
LIN {X 0,Y 591.917,Z 1130.829,A -85,B 0,C 180,E1 28468.009,E2 28468.009} C_VEL
LIN {X 0,Y 591.905,Z 1131.878,A -85,B 0,C 180,E1 28465.624,E2 28465.624} C_VEL
LIN {X 0,Y 591.871,Z 1131.551,A -85,B 0,C 180,E1 28463.075,E2 28463.075} C_VEL
LIN {X 0,Y 591.918,Z 1129.672,A -85,B 0,C 180,E1 28460.571,E2 28460.571} C_VEL
LIN {X 0,Y 591.951,Z 1126.145,A -85,B 0,C 180,E1 28458.006,E2 28458.006} C_VEL
LIN {X 0,Y 592.06,Z 1120.855,A -85,B 0,C 180,E1 28455.354,E2 28455.354} C_VEL
LIN {X 0,Y 592.261,Z 1113.726,A -85,B 0,C 180,E1 28452.678,E2 28452.678} C_VEL
LIN {X 0,Y 592.654,Z 1105.844,A -85,B 0,C 180,E1 28450.302,E2 28450.302} C_VEL
LIN {X 0,Y 593.264,Z 1095.563,A -85,B 0,C 180,E1 28447.692,E2 28447.692} C_VEL
LIN {X 0,Y 594.185,Z 1083.515,A -85,B 0,C 180,E1 28445.117,E2 28445.117} C_VEL
LIN {X 0,Y 595.29,Z 1071.502,A -85,B 0,C 180,E1 28442.888,E2 28442.888} C_VEL
LIN {X 0,Y 596.827,Z 1056.721,A -85,B 0,C 180,E1 28440.48,E2 28440.48} C_VEL
LIN {X 0,Y 598.743,Z 1039.933,A -85,B 0,C 180,E1 28438.086,E2 28438.086} C_VEL
LIN {X 0,Y 600.823,Z 1023.347,A -85,B 0,C 180,E1 28435.992,E2 28435.992} C_VEL
LIN {X 0,Y 603.353,Z 1003.844,A -85,B 0,C 180,E1 28433.816,E2 28433.816} C_VEL
LIN {X 0,Y 606.127,Z 983.244,A -85,B 0,C 180,E1 28431.796,E2 28431.796} C_VEL
LIN {X 0,Y 609.174,Z 961.084,A -85,B 0,C 180,E1 28429.885,E2 28429.885} C_VEL
LIN {X 0,Y 612.129,Z 939.128,A -85,B 0,C 180,E1 28428.218,E2 28428.218} C_VEL
LIN {X 0,Y 615.189,Z 915.443,A -85,B 0,C 180,E1 28426.656,E2 28426.656} C_VEL
LIN {X 0,Y 618.153,Z 891.435,A -85,B 0,C 180,E1 28425.288,E2 28425.288} C_VEL
LIN {X 0,Y 621.019,Z 866.448,A -85,B 0,C 180,E1 28424.067,E2 28424.067} C_VEL
LIN {X 0,Y 623.432,Z 842.561,A -85,B 0,C 180,E1 28423.076,E2 28423.076} C_VEL
LIN {X 0,Y 625.773,Z 816.225,A -85,B 0,C 180,E1 28422.176,E2 28422.176} C_VEL
LIN {X 0,Y 627.665,Z 791.387,A -85,B 0,C 180,E1 28421.493,E2 28421.493} C_VEL
LIN {X 0,Y 629.012,Z 765.511,A -85,B 0,C 180,E1 28420.969,E2 28420.969} C_VEL
LIN {X 0,Y 630.019,Z 730.123,A -85,B 0,C 180,E1 28420.462,E2 28420.462} C_VEL
LIN {X 0,Y 633.822,Z 533.239,A -85,B 0,C 180,E1 28417.841,E2 28417.841} C_VEL
LIN {X 0,Y 637.199,Z 412.164,A -85,B 0,C 180,E1 28416.112,E2 28416.112} C_VEL
LIN {X 0,Y 637.221,Z 407.708,A -85,B 0,C 180,E1 28416.033,E2 28416.033} C_VEL
LIN {X 0,Y 625.189,Z 389.651,A -85,B 0,C 180,E1 28414.305,E2 28414.305} C_VEL
LIN {X 0,Y 618.975,Z 380.409,A -85,B 0,C 180,E1 28413.198,E2 28413.198} C_VEL
LIN {X 0,Y 616.358,Z 376.604,A -85,B 0,C 180,E1 28412.654,E2 28412.654} C_VEL
LIN {X 0,Y 613.19,Z 371.982,A -85,B 0,C 180,E1 28411.904,E2 28411.904} C_VEL
LIN {X 0,Y 610.475,Z 368.247,A -85,B 0,C 180,E1 28411.107,E2 28411.107} C_VEL
LIN {X 0,Y 609.787,Z 366.98,A -85,B 0,C 180,E1 28410.856,E2 28410.856} C_VEL
LIN {X 0,Y 607.097,Z 364.441,A -85,B 0,C 180,E1 28409.657,E2 28409.657} C_VEL
LIN {X 0,Y 606.518,Z 363.229,A -85,B 0,C 180,E1 28409.009,E2 28409.009} C_VEL
LIN {X 0,Y 606.064,Z 365.312,A -85,B 0,C 180,E1 28408.078,E2 28408.078} C_VEL
LIN {X 0,Y 606.612,Z 368.889,A -85,B 0,C 180,E1 28407.103,E2 28407.103} C_VEL
LIN {X 0,Y 608.365,Z 374.456,A -85,B 0,C 180,E1 28406.083,E2 28406.083} C_VEL
LIN {X 0,Y 611.086,Z 381.206,A -85,B 0,C 180,E1 28405.119,E2 28405.119} C_VEL
LIN {X 0,Y 615.061,Z 390.715,A -85,B 0,C 180,E1 28404.065,E2 28404.065} C_VEL
LIN {X 0,Y 622.596,Z 407.682,A -85,B 0,C 180,E1 28402.564,E2 28402.564} C_VEL
LIN {X 0,Y 627.581,Z 416.407,A -85,B 0,C 180,E1 28401.79,E2 28401.79} C_VEL
LIN {X 0,Y 633.32,Z 453.076,A -85,B 0,C 180,E1 28400.494,E2 28400.494} C_VEL
LIN {X 0,Y 636.645,Z 469.873,A -85,B 0,C 180,E1 28399.894,E2 28399.894} C_VEL
LIN {X 0,Y 633.77,Z 604.148,A -85,B 0,C 180,E1 28398.016,E2 28398.016} C_VEL
LIN {X 0,Y 630.914,Z 796.724,A -85,B 0,C 180,E1 28395.518,E2 28395.518} C_VEL
LIN {X 0,Y 629.313,Z 904.022,A -85,B 0,C 180,E1 28394.153,E2 28394.153} C_VEL
LIN {X 0,Y 628.361,Z 928.436,A -85,B 0,C 180,E1 28393.741,E2 28393.741} C_VEL
LIN {X 0,Y 626.648,Z 955.148,A -85,B 0,C 180,E1 28393.103,E2 28393.103} C_VEL
LIN {X 0,Y 624.735,Z 978.137,A -85,B 0,C 180,E1 28392.392,E2 28392.392} C_VEL
LIN {X 0,Y 622.833,Z 998.279,A -85,B 0,C 180,E1 28391.653,E2 28391.653} C_VEL
LIN {X 0,Y 620.753,Z 1018.448,A -85,B 0,C 180,E1 28390.794,E2 28390.794} C_VEL
LIN {X 0,Y 618.547,Z 1038.062,A -85,B 0,C 180,E1 28389.839,E2 28389.839} C_VEL
LIN {X 0,Y 615.912,Z 1059.937,A -85,B 0,C 180,E1 28388.629,E2 28388.629} C_VEL
LIN {X 0,Y 612.644,Z 1084.843,A -85,B 0,C 180,E1 28387.03,E2 28387.03} C_VEL
LIN {X 0,Y 610.045,Z 1104.186,A -85,B 0,C 180,E1 28385.613,E2 28385.613} C_VEL
LIN {X 0,Y 607.591,Z 1122.331,A -85,B 0,C 180,E1 28384.129,E2 28384.129} C_VEL
LIN {X 0,Y 604.725,Z 1143.792,A -85,B 0,C 180,E1 28382.159,E2 28382.159} C_VEL
LIN {X 0,Y 602.2,Z 1162.447,A -85,B 0,C 180,E1 28380.205,E2 28380.205} C_VEL
LIN {X 0,Y 600.141,Z 1178.369,A -85,B 0,C 180,E1 28378.348,E2 28378.348} C_VEL
LIN {X 0,Y 598.086,Z 1195.735,A -85,B 0,C 180,E1 28376.083,E2 28376.083} C_VEL
LIN {X 0,Y 596.271,Z 1211.597,A -85,B 0,C 180,E1 28373.71,E2 28373.71} C_VEL
LIN {X 0,Y 595.066,Z 1223.611,A -85,B 0,C 180,E1 28371.688,E2 28371.688} C_VEL
LIN {X 0,Y 593.932,Z 1236.893,A -85,B 0,C 180,E1 28369.164,E2 28369.164} C_VEL
LIN {X 0,Y 593.093,Z 1248.086,A -85,B 0,C 180,E1 28366.654,E2 28366.654} C_VEL
LIN {X 0,Y 592.618,Z 1256.16,A -85,B 0,C 180,E1 28364.56,E2 28364.56} C_VEL
LIN {X 0,Y 592.293,Z 1263.052,A -85,B 0,C 180,E1 28362.479,E2 28362.479} C_VEL
LIN {X 0,Y 592.105,Z 1269.073,A -85,B 0,C 180,E1 28360.311,E2 28360.311} C_VEL
LIN {X 0,Y 591.948,Z 1274.735,A -85,B 0,C 180,E1 28357.766,E2 28357.766} C_VEL
LIN {X 0,Y 591.921,Z 1278.661,A -85,B 0,C 180,E1 28355.234,E2 28355.234} C_VEL
LIN {X 0,Y 591.91,Z 1280.812,A -85,B 0,C 180,E1 28353.002,E2 28353.002} C_VEL
LIN {X 0,Y 591.878,Z 1281.759,A -85,B 0,C 180,E1 28351.065,E2 28351.065} C_VEL
LIN {X 0,Y 591.868,Z 1281.804,A -85,B 0,C 180,E1 28349.129,E2 28349.129} C_VEL
LIN {X 0,Y 591.909,Z 1280.947,A -85,B 0,C 180,E1 28347.192,E2 28347.192} C_VEL
LIN {X 0,Y 591.92,Z 1279,A -85,B 0,C 180,E1 28345.058,E2 28345.058} C_VEL
LIN {X 0,Y 591.951,Z 1275.422,A -85,B 0,C 180,E1 28342.624,E2 28342.624} C_VEL
LIN {X 0,Y 592.067,Z 1269.836,A -85,B 0,C 180,E1 28339.983,E2 28339.983} C_VEL
LIN {X 0,Y 592.266,Z 1263.656,A -85,B 0,C 180,E1 28337.718,E2 28337.718} C_VEL
LIN {X 0,Y 592.591,Z 1256.51,A -85,B 0,C 180,E1 28335.539,E2 28335.539} C_VEL
LIN {X 0,Y 593.07,Z 1248.493,A -85,B 0,C 180,E1 28333.446,E2 28333.446} C_VEL
LIN {X 0,Y 593.838,Z 1237.83,A -85,B 0,C 180,E1 28331.037,E2 28331.037} C_VEL
LIN {X 0,Y 594.963,Z 1224.724,A -85,B 0,C 180,E1 28328.508,E2 28328.508} C_VEL
LIN {X 0,Y 596.223,Z 1212.1,A -85,B 0,C 180,E1 28326.371,E2 28326.371} C_VEL
LIN {X 0,Y 597.81,Z 1197.865,A -85,B 0,C 180,E1 28324.223,E2 28324.223} C_VEL
LIN {X 0,Y 599.968,Z 1179.895,A -85,B 0,C 180,E1 28321.839,E2 28321.839} C_VEL
LIN {X 0,Y 602.067,Z 1163.372,A -85,B 0,C 180,E1 28319.898,E2 28319.898} C_VEL
LIN {X 0,Y 604.299,Z 1146.749,A -85,B 0,C 180,E1 28318.142,E2 28318.142} C_VEL
LIN {X 0,Y 607.35,Z 1124.343,A -85,B 0,C 180,E1 28316.043,E2 28316.043} C_VEL
LIN {X 0,Y 609.907,Z 1105.218,A -85,B 0,C 180,E1 28314.468,E2 28314.468} C_VEL
LIN {X 0,Y 612.445,Z 1086.302,A -85,B 0,C 180,E1 28313.073,E2 28313.073} C_VEL
LIN {X 0,Y 615.459,Z 1063.493,A -85,B 0,C 180,E1 28311.581,E2 28311.581} C_VEL
LIN {X 0,Y 618.359,Z 1039.699,A -85,B 0,C 180,E1 28310.244,E2 28310.244} C_VEL
LIN {X 0,Y 620.678,Z 1019.138,A -85,B 0,C 180,E1 28309.237,E2 28309.237} C_VEL
LIN {X 0,Y 622.703,Z 999.562,A -85,B 0,C 180,E1 28308.398,E2 28308.398} C_VEL
LIN {X 0,Y 624.664,Z 978.876,A -85,B 0,C 180,E1 28307.633,E2 28307.633} C_VEL
LIN {X 0,Y 626.528,Z 956.585,A -85,B 0,C 180,E1 28306.938,E2 28306.938} C_VEL
LIN {X 0,Y 628.306,Z 930.169,A -85,B 0,C 180,E1 28306.291,E2 28306.291} C_VEL
LIN {X 0,Y 629.507,Z 903.849,A -85,B 0,C 180,E1 28305.824,E2 28305.824} C_VEL
LIN {X 0,Y 633.158,Z 735.24,A -85,B 0,C 180,E1 28303.548,E2 28303.548} C_VEL
LIN {X 0,Y 638.053,Z 536.367,A -85,B 0,C 180,E1 28300.774,E2 28300.774} C_VEL
LIN {X 0,Y 639.648,Z 469.001,A -85,B 0,C 180,E1 28299.801,E2 28299.801} C_VEL
LIN {X 0,Y 630.442,Z 419.846,A -85,B 0,C 180,E1 28297.879,E2 28297.879} C_VEL
LIN {X 0,Y 619.774,Z 397.512,A -85,B 0,C 180,E1 28294.941,E2 28294.941} C_VEL
LIN {X 0,Y 610.657,Z 379.891,A -85,B 0,C 180,E1 28292.34,E2 28292.34} C_VEL
LIN {X 0,Y 603.644,Z 366.74,A -85,B 0,C 180,E1 28290.235,E2 28290.235} C_VEL
LIN {X 0,Y 600.173,Z 360.763,A -85,B 0,C 180,E1 28289.194,E2 28289.194} C_VEL
LIN {X 0,Y 598.238,Z 356.98,A -85,B 0,C 180,E1 28288.556,E2 28288.556} C_VEL
LIN {X 0,Y 596.146,Z 353.23,A -85,B 0,C 180,E1 28287.883,E2 28287.883} C_VEL
LIN {X 0,Y 593.525,Z 348.822,A -85,B 0,C 180,E1 28287.056,E2 28287.056} C_VEL
LIN {X 0,Y 593.213,Z 347.534,A -85,B 0,C 180,E1 28286.801,E2 28286.801} C_VEL
LIN {X 0,Y 593.191,Z 347.326,A -85,B 0,C 180,E1 28283.546,E2 28283.546} C_VEL
LIN {X 0,Y 593.173,Z 347.333,A -85,B 0,C 180,E1 28280.411,E2 28280.411} C_VEL
LIN {X 0,Y 593.19,Z 347.333,A -85,B 0,C 180,E1 28277.258,E2 28277.258} C_VEL
LIN {X 0,Y 593.168,Z 347.341,A -85,B 0,C 180,E1 28274.048,E2 28274.048} C_VEL
LIN {X 0,Y 593.193,Z 347.333,A -85,B 0,C 180,E1 28270.882,E2 28270.882} C_VEL
LIN {X 0,Y 593.17,Z 347.34,A -85,B 0,C 180,E1 28267.653,E2 28267.653} C_VEL
LIN {X 0,Y 593.188,Z 347.332,A -85,B 0,C 180,E1 28264.35,E2 28264.35} C_VEL
LIN {X 0,Y 593.192,Z 347.327,A -85,B 0,C 180,E1 28261.062,E2 28261.062} C_VEL
LIN {X 0,Y 593.164,Z 347.342,A -85,B 0,C 180,E1 28257.778,E2 28257.778} C_VEL
LIN {X 0,Y 593.195,Z 347.336,A -85,B 0,C 180,E1 28254.584,E2 28254.584} C_VEL
LIN {X 0,Y 593.158,Z 347.34,A -85,B 0,C 180,E1 28251.469,E2 28251.469} C_VEL
LIN {X 0,Y 593.198,Z 347.339,A -85,B 0,C 180,E1 28248.326,E2 28248.326} C_VEL
LIN {X 0,Y 593.154,Z 347.341,A -85,B 0,C 180,E1 28245.153,E2 28245.153} C_VEL
LIN {X 0,Y 593.198,Z 347.335,A -85,B 0,C 180,E1 28241.927,E2 28241.927} C_VEL
LIN {X 0,Y 593.159,Z 347.34,A -85,B 0,C 180,E1 28238.751,E2 28238.751} C_VEL
LIN {X 0,Y 593.184,Z 347.342,A -85,B 0,C 180,E1 28235.502,E2 28235.502} C_VEL
LIN {X 0,Y 593.166,Z 347.339,A -85,B 0,C 180,E1 28232.383,E2 28232.383} C_VEL
LIN {X 0,Y 593.16,Z 347.345,A -85,B 0,C 180,E1 28229.06,E2 28229.06} C_VEL
LIN {X 0,Y 593.182,Z 347.338,A -85,B 0,C 180,E1 28225.969,E2 28225.969} C_VEL
LIN {X 0,Y 593.148,Z 347.345,A -85,B 0,C 180,E1 28222.717,E2 28222.717} C_VEL
LIN {X 0,Y 593.199,Z 347.337,A -85,B 0,C 180,E1 28219.63,E2 28219.63} C_VEL
LIN {X 0,Y 593.143,Z 347.344,A -85,B 0,C 180,E1 28216.411,E2 28216.411} C_VEL
LIN {X 0,Y 593.201,Z 347.339,A -85,B 0,C 180,E1 28213.266,E2 28213.266} C_VEL
LIN {X 0,Y 593.139,Z 347.345,A -85,B 0,C 180,E1 28210.213,E2 28210.213} C_VEL
LIN {X 0,Y 593.198,Z 347.339,A -85,B 0,C 180,E1 28207.116,E2 28207.116} C_VEL
LIN {X 0,Y 593.134,Z 347.345,A -85,B 0,C 180,E1 28203.962,E2 28203.962} C_VEL
LIN {X 0,Y 593.204,Z 347.34,A -85,B 0,C 180,E1 28200.824,E2 28200.824} C_VEL
LIN {X 0,Y 593.13,Z 347.343,A -85,B 0,C 180,E1 28197.728,E2 28197.728} C_VEL
LIN {X 0,Y 593.164,Z 347.339,A -85,B 0,C 180,E1 28195.045,E2 28195.045} C_VEL
LIN {X 0,Y 592.224,Z 347.462,A -85,B 0,C 180,E1 28194.3,E2 28194.3} C_VEL
LIN {X 0,Y 585.643,Z 348.281,A -85,B 0,C 180,E1 28192.159,E2 28192.159} C_VEL
LIN {X 0,Y 585.189,Z 348.332,A -85,B 0,C 180,E1 28191.669,E2 28191.669} C_VEL
LIN {X 0,Y 585.249,Z 348.329,A -85,B 0,C 180,E1 28188.632,E2 28188.632} C_VEL
LIN {X 0,Y 585.184,Z 348.328,A -85,B 0,C 180,E1 28185.459,E2 28185.459} C_VEL
LIN {X 0,Y 585.233,Z 348.325,A -85,B 0,C 180,E1 28182.532,E2 28182.532} C_VEL
LIN {X 0,Y 585.182,Z 348.335,A -85,B 0,C 180,E1 28179.342,E2 28179.342} C_VEL
LIN {X 0,Y 585.227,Z 348.331,A -85,B 0,C 180,E1 28176.376,E2 28176.376} C_VEL
LIN {X 0,Y 585.178,Z 348.334,A -85,B 0,C 180,E1 28173.134,E2 28173.134} C_VEL
LIN {X 0,Y 585.249,Z 348.324,A -85,B 0,C 180,E1 28170,E2 28170} C_VEL
LIN {X 0,Y 585.167,Z 348.304,A -85,B 0,C 180,E1 28166.866,E2 28166.866} C_VEL
LIN {X 0,Y 585.248,Z 348.3,A -85,B 0,C 180,E1 28163.723,E2 28163.723} C_VEL
LIN {X 0,Y 585.286,Z 348.588,A -85,B 0,C 180,E1 28161.7,E2 28161.7} C_VEL
LIN {X 0,Y 585.723,Z 350.262,A -85,B 0,C 180,E1 28161.459,E2 28161.459} C_VEL
LIN {X 0,Y 587.652,Z 353.182,A -85,B 0,C 180,E1 28161.118,E2 28161.118} C_VEL
LIN {X 0,Y 589.786,Z 354.923,A -85,B 0,C 180,E1 28160.781,E2 28160.781} C_VEL
LIN {X 0,Y 592.243,Z 358.733,A -85,B 0,C 180,E1 28160.351,E2 28160.351} C_VEL
LIN {X 0,Y 594.522,Z 361.009,A -85,B 0,C 180,E1 28159.988,E2 28159.988} C_VEL
LIN {X 0,Y 597.687,Z 365.255,A -85,B 0,C 180,E1 28159.469,E2 28159.469} C_VEL
LIN {X 0,Y 599.558,Z 367.671,A -85,B 0,C 180,E1 28159.17,E2 28159.17} C_VEL
LIN {X 0,Y 604.063,Z 373.401,A -85,B 0,C 180,E1 28158.468,E2 28158.468} C_VEL
LIN {X 0,Y 615.237,Z 387.714,A -85,B 0,C 180,E1 28156.825,E2 28156.825} C_VEL
LIN {X 0,Y 627.02,Z 403.977,A -85,B 0,C 180,E1 28155.183,E2 28155.183} C_VEL
LIN {X 0,Y 632.84,Z 412.313,A -85,B 0,C 180,E1 28154.421,E2 28154.421} C_VEL
LIN {X 0,Y 627.017,Z 621.074,A -85,B 0,C 180,E1 28151.468,E2 28151.468} C_VEL
LIN {X 0,Y 623.556,Z 758.95,A -85,B 0,C 180,E1 28149.564,E2 28149.564} C_VEL
LIN {X 0,Y 622.052,Z 786.188,A -85,B 0,C 180,E1 28149.036,E2 28149.036} C_VEL
LIN {X 0,Y 620.149,Z 812.071,A -85,B 0,C 180,E1 28148.36,E2 28148.36} C_VEL
LIN {X 0,Y 617.974,Z 836.781,A -85,B 0,C 180,E1 28147.552,E2 28147.552} C_VEL
LIN {X 0,Y 615.528,Z 860.475,A -85,B 0,C 180,E1 28146.609,E2 28146.609} C_VEL
LIN {X 0,Y 612.804,Z 883.674,A -85,B 0,C 180,E1 28145.516,E2 28145.516} C_VEL
LIN {X 0,Y 609.903,Z 906.93,A -85,B 0,C 180,E1 28144.25,E2 28144.25} C_VEL
LIN {X 0,Y 606.854,Z 929.262,A -85,B 0,C 180,E1 28142.841,E2 28142.841} C_VEL
LIN {X 0,Y 603.472,Z 953.058,A -85,B 0,C 180,E1 28141.12,E2 28141.12} C_VEL
LIN {X 0,Y 600.432,Z 974.332,A -85,B 0,C 180,E1 28139.365,E2 28139.365} C_VEL
LIN {X 0,Y 597.375,Z 995.786,A -85,B 0,C 180,E1 28137.344,E2 28137.344} C_VEL
LIN {X 0,Y 594.639,Z 1014.744,A -85,B 0,C 180,E1 28135.312,E2 28135.312} C_VEL
LIN {X 0,Y 592.077,Z 1033.706,A -85,B 0,C 180,E1 28133.016,E2 28133.016} C_VEL
LIN {X 0,Y 589.889,Z 1050.842,A -85,B 0,C 180,E1 28130.659,E2 28130.659} C_VEL
LIN {X 0,Y 588.061,Z 1066.872,A -85,B 0,C 180,E1 28128.137,E2 28128.137} C_VEL
LIN {X 0,Y 586.62,Z 1080.949,A -85,B 0,C 180,E1 28125.577,E2 28125.577} C_VEL
LIN {X 0,Y 585.601,Z 1092.993,A -85,B 0,C 180,E1 28123.048,E2 28123.048} C_VEL
LIN {X 0,Y 584.807,Z 1103.771,A -85,B 0,C 180,E1 28120.392,E2 28120.392} C_VEL
LIN {X 0,Y 584.394,Z 1111.841,A -85,B 0,C 180,E1 28118.022,E2 28118.022} C_VEL
LIN {X 0,Y 584.101,Z 1119.065,A -85,B 0,C 180,E1 28115.43,E2 28115.43} C_VEL
LIN {X 0,Y 583.943,Z 1124.418,A -85,B 0,C 180,E1 28112.992,E2 28112.992} C_VEL
LIN {X 0,Y 583.93,Z 1128.301,A -85,B 0,C 180,E1 28110.538,E2 28110.538} C_VEL
LIN {X 0,Y 583.918,Z 1130.803,A -85,B 0,C 180,E1 28108.093,E2 28108.093} C_VEL
LIN {X 0,Y 583.906,Z 1131.871,A -85,B 0,C 180,E1 28105.674,E2 28105.674} C_VEL
LIN {X 0,Y 583.874,Z 1131.595,A -85,B 0,C 180,E1 28103.132,E2 28103.132} C_VEL
LIN {X 0,Y 583.918,Z 1129.714,A -85,B 0,C 180,E1 28100.551,E2 28100.551} C_VEL
LIN {X 0,Y 583.954,Z 1126.211,A -85,B 0,C 180,E1 28097.951,E2 28097.951} C_VEL
LIN {X 0,Y 584.071,Z 1121.007,A -85,B 0,C 180,E1 28095.286,E2 28095.286} C_VEL
LIN {X 0,Y 584.285,Z 1113.865,A -85,B 0,C 180,E1 28092.553,E2 28092.553} C_VEL
LIN {X 0,Y 584.703,Z 1106.01,A -85,B 0,C 180,E1 28090.145,E2 28090.145} C_VEL
LIN {X 0,Y 585.35,Z 1096.017,A -85,B 0,C 180,E1 28087.558,E2 28087.558} C_VEL
LIN {X 0,Y 586.309,Z 1084.273,A -85,B 0,C 180,E1 28084.99,E2 28084.99} C_VEL
LIN {X 0,Y 587.537,Z 1071.682,A -85,B 0,C 180,E1 28082.614,E2 28082.614} C_VEL
LIN {X 0,Y 589.246,Z 1056.425,A -85,B 0,C 180,E1 28080.097,E2 28080.097} C_VEL
LIN {X 0,Y 591.304,Z 1039.605,A -85,B 0,C 180,E1 28077.674,E2 28077.674} C_VEL
LIN {X 0,Y 593.653,Z 1022.206,A -85,B 0,C 180,E1 28075.46,E2 28075.46} C_VEL
LIN {X 0,Y 596.508,Z 1001.648,A -85,B 0,C 180,E1 28073.165,E2 28073.165} C_VEL
LIN {X 0,Y 599.433,Z 981.242,A -85,B 0,C 180,E1 28071.172,E2 28071.172} C_VEL
LIN {X 0,Y 602.662,Z 958.789,A -85,B 0,C 180,E1 28069.243,E2 28069.243} C_VEL
LIN {X 0,Y 605.832,Z 936.483,A -85,B 0,C 180,E1 28067.562,E2 28067.562} C_VEL
LIN {X 0,Y 609.163,Z 912.468,A -85,B 0,C 180,E1 28065.989,E2 28065.989} C_VEL
LIN {X 0,Y 612.079,Z 889.654,A -85,B 0,C 180,E1 28064.703,E2 28064.703} C_VEL
LIN {X 0,Y 614.98,Z 865.31,A -85,B 0,C 180,E1 28063.518,E2 28063.518} C_VEL
LIN {X 0,Y 617.403,Z 842.374,A -85,B 0,C 180,E1 28062.566,E2 28062.566} C_VEL
LIN {X 0,Y 619.656,Z 816.815,A -85,B 0,C 180,E1 28061.702,E2 28061.702} C_VEL
LIN {X 0,Y 621.423,Z 792.102,A -85,B 0,C 180,E1 28061.039,E2 28061.039} C_VEL
LIN {X 0,Y 622.787,Z 766.397,A -85,B 0,C 180,E1 28060.516,E2 28060.516} C_VEL
LIN {X 0,Y 623.82,Z 728.533,A -85,B 0,C 180,E1 28059.979,E2 28059.979} C_VEL
LIN {X 0,Y 627.587,Z 549.371,A -85,B 0,C 180,E1 28057.565,E2 28057.565} C_VEL
LIN {X 0,Y 631.266,Z 428.617,A -85,B 0,C 180,E1 28055.816,E2 28055.816} C_VEL
LIN {X 0,Y 631.849,Z 411.742,A -85,B 0,C 180,E1 28055.548,E2 28055.548} C_VEL
LIN {X 0,Y 621.362,Z 395.487,A -85,B 0,C 180,E1 28053.932,E2 28053.932} C_VEL
LIN {X 0,Y 615.599,Z 386.651,A -85,B 0,C 180,E1 28052.844,E2 28052.844} C_VEL
LIN {X 0,Y 613.202,Z 383.071,A -85,B 0,C 180,E1 28052.301,E2 28052.301} C_VEL
LIN {X 0,Y 610.581,Z 379.037,A -85,B 0,C 180,E1 28051.62,E2 28051.62} C_VEL
LIN {X 0,Y 607.957,Z 374.907,A -85,B 0,C 180,E1 28050.76,E2 28050.76} C_VEL
LIN {X 0,Y 605.424,Z 372.051,A -85,B 0,C 180,E1 28049.479,E2 28049.479} C_VEL
LIN {X 0,Y 605.04,Z 371.203,A -85,B 0,C 180,E1 28049.058,E2 28049.058} C_VEL
LIN {X 0,Y 604.514,Z 372.936,A -85,B 0,C 180,E1 28048.265,E2 28048.265} C_VEL
LIN {X 0,Y 604.773,Z 376.102,A -85,B 0,C 180,E1 28047.385,E2 28047.385} C_VEL
LIN {X 0,Y 605.961,Z 381.125,A -85,B 0,C 180,E1 28046.437,E2 28046.437} C_VEL
LIN {X 0,Y 608.421,Z 388.236,A -85,B 0,C 180,E1 28045.403,E2 28045.403} C_VEL
LIN {X 0,Y 611.641,Z 396.635,A -85,B 0,C 180,E1 28044.453,E2 28044.453} C_VEL
LIN {X 0,Y 617.941,Z 412.034,A -85,B 0,C 180,E1 28043.055,E2 28043.055} C_VEL
LIN {X 0,Y 622.763,Z 420.94,A -85,B 0,C 180,E1 28042.235,E2 28042.235} C_VEL
LIN {X 0,Y 627.977,Z 456.318,A -85,B 0,C 180,E1 28040.947,E2 28040.947} C_VEL
LIN {X 0,Y 630.897,Z 471.851,A -85,B 0,C 180,E1 28040.377,E2 28040.377} C_VEL
LIN {X 0,Y 627.629,Z 602.898,A -85,B 0,C 180,E1 28038.5,E2 28038.5} C_VEL
LIN {X 0,Y 624.75,Z 773.25,A -85,B 0,C 180,E1 28036.243,E2 28036.243} C_VEL
LIN {X 0,Y 622.745,Z 901.288,A -85,B 0,C 180,E1 28034.601,E2 28034.601} C_VEL
LIN {X 0,Y 621.686,Z 927.7,A -85,B 0,C 180,E1 28034.158,E2 28034.158} C_VEL
LIN {X 0,Y 620.001,Z 956.81,A -85,B 0,C 180,E1 28033.491,E2 28033.491} C_VEL
LIN {X 0,Y 618.593,Z 978.005,A -85,B 0,C 180,E1 28032.882,E2 28032.882} C_VEL
LIN {X 0,Y 617.037,Z 995.701,A -85,B 0,C 180,E1 28032.259,E2 28032.259} C_VEL
LIN {X 0,Y 614.819,Z 1016.44,A -85,B 0,C 180,E1 28031.383,E2 28031.383} C_VEL
LIN {X 0,Y 612.607,Z 1035.136,A -85,B 0,C 180,E1 28030.483,E2 28030.483} C_VEL
LIN {X 0,Y 610.251,Z 1053.721,A -85,B 0,C 180,E1 28029.474,E2 28029.474} C_VEL
LIN {X 0,Y 607.666,Z 1073.103,A -85,B 0,C 180,E1 28028.29,E2 28028.29} C_VEL
LIN {X 0,Y 604.561,Z 1095.841,A -85,B 0,C 180,E1 28026.718,E2 28026.718} C_VEL
LIN {X 0,Y 601.294,Z 1118.166,A -85,B 0,C 180,E1 28024.934,E2 28024.934} C_VEL
LIN {X 0,Y 598.803,Z 1135.366,A -85,B 0,C 180,E1 28023.393,E2 28023.393} C_VEL
LIN {X 0,Y 596.375,Z 1152.323,A -85,B 0,C 180,E1 28021.709,E2 28021.709} C_VEL
LIN {X 0,Y 593.565,Z 1172.67,A -85,B 0,C 180,E1 28019.435,E2 28019.435} C_VEL
LIN {X 0,Y 591.38,Z 1188.841,A -85,B 0,C 180,E1 28017.38,E2 28017.38} C_VEL
LIN {X 0,Y 589.592,Z 1203.342,A -85,B 0,C 180,E1 28015.322,E2 28015.322} C_VEL
LIN {X 0,Y 587.778,Z 1219.54,A -85,B 0,C 180,E1 28012.715,E2 28012.715} C_VEL
LIN {X 0,Y 586.548,Z 1231.753,A -85,B 0,C 180,E1 28010.454,E2 28010.454} C_VEL
LIN {X 0,Y 585.642,Z 1241.987,A -85,B 0,C 180,E1 28008.309,E2 28008.309} C_VEL
LIN {X 0,Y 584.933,Z 1252.137,A -85,B 0,C 180,E1 28005.873,E2 28005.873} C_VEL
LIN {X 0,Y 584.421,Z 1261.532,A -85,B 0,C 180,E1 28003.153,E2 28003.153} C_VEL
LIN {X 0,Y 584.145,Z 1267.802,A -85,B 0,C 180,E1 28000.953,E2 28000.953} C_VEL
LIN {X 0,Y 584.013,Z 1273.132,A -85,B 0,C 180,E1 27998.665,E2 27998.665} C_VEL
LIN {X 0,Y 583.94,Z 1277.634,A -85,B 0,C 180,E1 27996.094,E2 27996.094} C_VEL
LIN {X 0,Y 583.912,Z 1280.472,A -85,B 0,C 180,E1 27993.534,E2 27993.534} C_VEL
LIN {X 0,Y 583.895,Z 1281.714,A -85,B 0,C 180,E1 27991.276,E2 27991.276} C_VEL
LIN {X 0,Y 583.865,Z 1281.827,A -85,B 0,C 180,E1 27989.215,E2 27989.215} C_VEL
LIN {X 0,Y 583.908,Z 1281.015,A -85,B 0,C 180,E1 27987.252,E2 27987.252} C_VEL
LIN {X 0,Y 583.92,Z 1279.111,A -85,B 0,C 180,E1 27985.088,E2 27985.088} C_VEL
LIN {X 0,Y 583.958,Z 1275.744,A -85,B 0,C 180,E1 27982.721,E2 27982.721} C_VEL
LIN {X 0,Y 584.05,Z 1270.595,A -85,B 0,C 180,E1 27980.143,E2 27980.143} C_VEL
LIN {X 0,Y 584.301,Z 1263.656,A -85,B 0,C 180,E1 27977.548,E2 27977.548} C_VEL
LIN {X 0,Y 584.666,Z 1256.509,A -85,B 0,C 180,E1 27975.339,E2 27975.339} C_VEL
LIN {X 0,Y 585.163,Z 1248.492,A -85,B 0,C 180,E1 27973.216,E2 27973.216} C_VEL
LIN {X 0,Y 585.963,Z 1238.297,A -85,B 0,C 180,E1 27970.875,E2 27970.875} C_VEL
LIN {X 0,Y 587.214,Z 1224.722,A -85,B 0,C 180,E1 27968.21,E2 27968.21} C_VEL
LIN {X 0,Y 588.537,Z 1212.25,A -85,B 0,C 180,E1 27966.069,E2 27966.069} C_VEL
LIN {X 0,Y 590.179,Z 1198.577,A -85,B 0,C 180,E1 27963.973,E2 27963.973} C_VEL
LIN {X 0,Y 592.54,Z 1180.057,A -85,B 0,C 180,E1 27961.475,E2 27961.475} C_VEL
LIN {X 0,Y 594.76,Z 1163.833,A -85,B 0,C 180,E1 27959.545,E2 27959.545} C_VEL
LIN {X 0,Y 597.036,Z 1147.762,A -85,B 0,C 180,E1 27957.821,E2 27957.821} C_VEL
LIN {X 0,Y 600.058,Z 1127.11,A -85,B 0,C 180,E1 27955.837,E2 27955.837} C_VEL
LIN {X 0,Y 603.041,Z 1105.883,A -85,B 0,C 180,E1 27954.059,E2 27954.059} C_VEL
LIN {X 0,Y 605.715,Z 1087.034,A -85,B 0,C 180,E1 27952.653,E2 27952.653} C_VEL
LIN {X 0,Y 608.511,Z 1066.811,A -85,B 0,C 180,E1 27951.307,E2 27951.307} C_VEL
LIN {X 0,Y 611.941,Z 1040.7,A -85,B 0,C 180,E1 27949.804,E2 27949.804} C_VEL
LIN {X 0,Y 614.424,Z 1019.834,A -85,B 0,C 180,E1 27948.771,E2 27948.771} C_VEL
LIN {X 0,Y 616.631,Z 999.559,A -85,B 0,C 180,E1 27947.895,E2 27947.895} C_VEL
LIN {X 0,Y 618.219,Z 982.835,A -85,B 0,C 180,E1 27947.275,E2 27947.275} C_VEL
LIN {X 0,Y 619.992,Z 960.768,A -85,B 0,C 180,E1 27946.585,E2 27946.585} C_VEL
LIN {X 0,Y 621.518,Z 939.141,A -85,B 0,C 180,E1 27946.026,E2 27946.026} C_VEL
LIN {X 0,Y 622.831,Z 916.564,A -85,B 0,C 180,E1 27945.557,E2 27945.557} C_VEL
LIN {X 0,Y 624.04,Z 884.594,A -85,B 0,C 180,E1 27945.069,E2 27945.069} C_VEL
LIN {X 0,Y 628.635,Z 682.882,A -85,B 0,C 180,E1 27942.317,E2 27942.317} C_VEL
LIN {X 0,Y 632.671,Z 535.688,A -85,B 0,C 180,E1 27940.228,E2 27940.228} C_VEL
LIN {X 0,Y 634.34,Z 471.034,A -85,B 0,C 180,E1 27939.282,E2 27939.282} C_VEL
LIN {X 0,Y 625.64,Z 424.721,A -85,B 0,C 180,E1 27937.453,E2 27937.453} C_VEL
LIN {X 0,Y 621.346,Z 417.963,A -85,B 0,C 180,E1 27936.772,E2 27936.772} C_VEL
LIN {X 0,Y 612.263,Z 398.935,A -85,B 0,C 180,E1 27934.18,E2 27934.18} C_VEL
LIN {X 0,Y 603.387,Z 381.81,A -85,B 0,C 180,E1 27931.578,E2 27931.578} C_VEL
LIN {X 0,Y 597.49,Z 371.154,A -85,B 0,C 180,E1 27929.803,E2 27929.803} C_VEL
LIN {X 0,Y 595.09,Z 366.758,A -85,B 0,C 180,E1 27929.051,E2 27929.051} C_VEL
LIN {X 0,Y 592.726,Z 362.436,A -85,B 0,C 180,E1 27928.289,E2 27928.289} C_VEL
LIN {X 0,Y 590.13,Z 357.757,A -85,B 0,C 180,E1 27927.443,E2 27927.443} C_VEL
LIN {X 0,Y 588.191,Z 354.069,A -85,B 0,C 180,E1 27926.775,E2 27926.775} C_VEL
LIN {X 0,Y 585.567,Z 349.754,A -85,B 0,C 180,E1 27925.921,E2 27925.921} C_VEL
LIN {X 0,Y 585.28,Z 348.514,A -85,B 0,C 180,E1 27925.663,E2 27925.663} C_VEL
LIN {X 0,Y 585.234,Z 348.335,A -85,B 0,C 180,E1 27922.437,E2 27922.437} C_VEL
LIN {X 0,Y 585.252,Z 348.329,A -85,B 0,C 180,E1 27919.253,E2 27919.253} C_VEL
LIN {X 0,Y 585.231,Z 348.328,A -85,B 0,C 180,E1 27916.068,E2 27916.068} C_VEL
LIN {X 0,Y 585.254,Z 348.323,A -85,B 0,C 180,E1 27912.833,E2 27912.833} C_VEL
LIN {X 0,Y 585.242,Z 348.326,A -85,B 0,C 180,E1 27909.539,E2 27909.539} C_VEL
LIN {X 0,Y 585.236,Z 348.323,A -85,B 0,C 180,E1 27906.179,E2 27906.179} C_VEL
LIN {X 0,Y 585.255,Z 348.329,A -85,B 0,C 180,E1 27902.938,E2 27902.938} C_VEL
LIN {X 0,Y 585.224,Z 348.332,A -85,B 0,C 180,E1 27899.706,E2 27899.706} C_VEL
LIN {X 0,Y 585.257,Z 348.327,A -85,B 0,C 180,E1 27896.474,E2 27896.474} C_VEL
LIN {X 0,Y 585.224,Z 348.327,A -85,B 0,C 180,E1 27893.23,E2 27893.23} C_VEL
LIN {X 0,Y 585.251,Z 348.33,A -85,B 0,C 180,E1 27889.964,E2 27889.964} C_VEL
LIN {X 0,Y 585.238,Z 348.327,A -85,B 0,C 180,E1 27886.765,E2 27886.765} C_VEL
LIN {X 0,Y 585.223,Z 348.324,A -85,B 0,C 180,E1 27883.421,E2 27883.421} C_VEL
LIN {X 0,Y 585.258,Z 348.325,A -85,B 0,C 180,E1 27880.228,E2 27880.228} C_VEL
LIN {X 0,Y 585.213,Z 348.323,A -85,B 0,C 180,E1 27877.06,E2 27877.06} C_VEL
LIN {X 0,Y 585.261,Z 348.323,A -85,B 0,C 180,E1 27873.846,E2 27873.846} C_VEL
LIN {X 0,Y 585.21,Z 348.323,A -85,B 0,C 180,E1 27870.747,E2 27870.747} C_VEL
LIN {X 0,Y 585.259,Z 348.323,A -85,B 0,C 180,E1 27867.557,E2 27867.557} C_VEL
LIN {X 0,Y 585.207,Z 348.324,A -85,B 0,C 180,E1 27864.418,E2 27864.418} C_VEL
LIN {X 0,Y 585.251,Z 348.323,A -85,B 0,C 180,E1 27861.17,E2 27861.17} C_VEL
LIN {X 0,Y 585.211,Z 348.324,A -85,B 0,C 180,E1 27858.082,E2 27858.082} C_VEL
LIN {X 0,Y 585.224,Z 348.325,A -85,B 0,C 180,E1 27854.742,E2 27854.742} C_VEL
LIN {X 0,Y 585.219,Z 348.324,A -85,B 0,C 180,E1 27851.699,E2 27851.699} C_VEL
LIN {X 0,Y 585.212,Z 348.326,A -85,B 0,C 180,E1 27848.456,E2 27848.456} C_VEL
LIN {X 0,Y 585.226,Z 348.323,A -85,B 0,C 180,E1 27845.394,E2 27845.394} C_VEL
LIN {X 0,Y 585.199,Z 348.328,A -85,B 0,C 180,E1 27842.099,E2 27842.099} C_VEL
LIN {X 0,Y 585.231,Z 348.32,A -85,B 0,C 180,E1 27839.139,E2 27839.139} C_VEL
LIN {X 0,Y 585.196,Z 348.329,A -85,B 0,C 180,E1 27835.938,E2 27835.938} C_VEL
LIN {X 0,Y 585.23,Z 348.32,A -85,B 0,C 180,E1 27832.926,E2 27832.926} C_VEL
LIN {X 0,Y 585.189,Z 348.332,A -85,B 0,C 180,E1 27831.669,E2 27831.669} C_VEL
LIN {X 0,Y 584.211,Z 348.452,A -85,B 0,C 180,E1 27830.915,E2 27830.915} C_VEL
LIN {X 0,Y 577.775,Z 349.261,A -85,B 0,C 180,E1 27828.743,E2 27828.743} C_VEL
LIN {X 0,Y 577.302,Z 349.313,A -85,B 0,C 180,E1 27828.247,E2 27828.247} C_VEL
LIN {X 0,Y 577.246,Z 349.316,A -85,B 0,C 180,E1 27825.242,E2 27825.242} C_VEL
LIN {X 0,Y 577.305,Z 349.313,A -85,B 0,C 180,E1 27822.097,E2 27822.097} C_VEL
LIN {X 0,Y 577.241,Z 349.325,A -85,B 0,C 180,E1 27819.069,E2 27819.069} C_VEL
LIN {X 0,Y 577.308,Z 349.32,A -85,B 0,C 180,E1 27815.965,E2 27815.965} C_VEL
LIN {X 0,Y 577.238,Z 349.321,A -85,B 0,C 180,E1 27812.879,E2 27812.879} C_VEL
LIN {X 0,Y 577.296,Z 349.317,A -85,B 0,C 180,E1 27809.702,E2 27809.702} C_VEL
LIN {X 0,Y 577.232,Z 349.293,A -85,B 0,C 180,E1 27806.624,E2 27806.624} C_VEL
LIN {X 0,Y 577.278,Z 349.288,A -85,B 0,C 180,E1 27803.436,E2 27803.436} C_VEL
LIN {X 0,Y 577.276,Z 349.624,A -85,B 0,C 180,E1 27802.836,E2 27802.836} C_VEL
LIN {X 0,Y 577.771,Z 351.359,A -85,B 0,C 180,E1 27802.586,E2 27802.586} C_VEL
LIN {X 0,Y 579.765,Z 354.192,A -85,B 0,C 180,E1 27802.219,E2 27802.219} C_VEL
LIN {X 0,Y 581.922,Z 355.979,A -85,B 0,C 180,E1 27801.863,E2 27801.863} C_VEL
LIN {X 0,Y 584.286,Z 359.726,A -85,B 0,C 180,E1 27801.438,E2 27801.438} C_VEL
LIN {X 0,Y 586.713,Z 362.145,A -85,B 0,C 180,E1 27801.041,E2 27801.041} C_VEL
LIN {X 0,Y 589.896,Z 366.299,A -85,B 0,C 180,E1 27800.508,E2 27800.508} C_VEL
LIN {X 0,Y 591.489,Z 368.107,A -85,B 0,C 180,E1 27800.247,E2 27800.247} C_VEL
LIN {X 0,Y 601.05,Z 380.483,A -85,B 0,C 180,E1 27798.704,E2 27798.704} C_VEL
LIN {X 0,Y 611.675,Z 394.166,A -85,B 0,C 180,E1 27797.119,E2 27797.119} C_VEL
LIN {X 0,Y 623.321,Z 410.331,A -85,B 0,C 180,E1 27795.473,E2 27795.473} C_VEL
LIN {X 0,Y 627.437,Z 416.356,A -85,B 0,C 180,E1 27794.914,E2 27794.914} C_VEL
LIN {X 0,Y 621.255,Z 625.671,A -85,B 0,C 180,E1 27791.929,E2 27791.929} C_VEL
LIN {X 0,Y 617.667,Z 759.359,A -85,B 0,C 180,E1 27790.063,E2 27790.063} C_VEL
LIN {X 0,Y 616.111,Z 787.04,A -85,B 0,C 180,E1 27789.526,E2 27789.526} C_VEL
LIN {X 0,Y 614.148,Z 812.7,A -85,B 0,C 180,E1 27788.85,E2 27788.85} C_VEL
LIN {X 0,Y 611.977,Z 836.737,A -85,B 0,C 180,E1 27788.065,E2 27788.065} C_VEL
LIN {X 0,Y 609.231,Z 862.445,A -85,B 0,C 180,E1 27787.034,E2 27787.034} C_VEL
LIN {X 0,Y 606.32,Z 885.81,A -85,B 0,C 180,E1 27785.911,E2 27785.911} C_VEL
LIN {X 0,Y 602.973,Z 910.763,A -85,B 0,C 180,E1 27784.513,E2 27784.513} C_VEL
LIN {X 0,Y 599.712,Z 933.648,A -85,B 0,C 180,E1 27783.032,E2 27783.032} C_VEL
LIN {X 0,Y 596.277,Z 956.249,A -85,B 0,C 180,E1 27781.342,E2 27781.342} C_VEL
LIN {X 0,Y 592.904,Z 978.502,A -85,B 0,C 180,E1 27779.439,E2 27779.439} C_VEL
LIN {X 0,Y 589.758,Z 999.266,A -85,B 0,C 180,E1 27777.419,E2 27777.419} C_VEL
LIN {X 0,Y 586.886,Z 1018.331,A -85,B 0,C 180,E1 27775.317,E2 27775.317} C_VEL
LIN {X 0,Y 584.309,Z 1036.386,A -85,B 0,C 180,E1 27773.049,E2 27773.049} C_VEL
LIN {X 0,Y 582.006,Z 1053.355,A -85,B 0,C 180,E1 27770.634,E2 27770.634} C_VEL
LIN {X 0,Y 580.144,Z 1068.79,A -85,B 0,C 180,E1 27768.122,E2 27768.122} C_VEL
LIN {X 0,Y 578.776,Z 1081.598,A -85,B 0,C 180,E1 27765.738,E2 27765.738} C_VEL
LIN {X 0,Y 577.677,Z 1093.722,A -85,B 0,C 180,E1 27763.134,E2 27763.134} C_VEL
LIN {X 0,Y 576.838,Z 1104.462,A -85,B 0,C 180,E1 27760.413,E2 27760.413} C_VEL
LIN {X 0,Y 576.404,Z 1112.427,A -85,B 0,C 180,E1 27758.012,E2 27758.012} C_VEL
LIN {X 0,Y 576.111,Z 1119.215,A -85,B 0,C 180,E1 27755.514,E2 27755.514} C_VEL
LIN {X 0,Y 575.947,Z 1124.588,A -85,B 0,C 180,E1 27753.017,E2 27753.017} C_VEL
LIN {X 0,Y 575.932,Z 1128.371,A -85,B 0,C 180,E1 27750.559,E2 27750.559} C_VEL
LIN {X 0,Y 575.917,Z 1130.853,A -85,B 0,C 180,E1 27748.067,E2 27748.067} C_VEL
LIN {X 0,Y 575.904,Z 1131.883,A -85,B 0,C 180,E1 27745.615,E2 27745.615} C_VEL
LIN {X 0,Y 575.868,Z 1131.534,A -85,B 0,C 180,E1 27742.996,E2 27742.996} C_VEL
LIN {X 0,Y 575.917,Z 1129.648,A -85,B 0,C 180,E1 27740.424,E2 27740.424} C_VEL
LIN {X 0,Y 575.963,Z 1126.107,A -85,B 0,C 180,E1 27737.791,E2 27737.791} C_VEL
LIN {X 0,Y 576.091,Z 1120.864,A -85,B 0,C 180,E1 27735.091,E2 27735.091} C_VEL
LIN {X 0,Y 576.32,Z 1113.858,A -85,B 0,C 180,E1 27732.375,E2 27732.375} C_VEL
LIN {X 0,Y 576.752,Z 1106.174,A -85,B 0,C 180,E1 27729.984,E2 27729.984} C_VEL
LIN {X 0,Y 577.458,Z 1096.222,A -85,B 0,C 180,E1 27727.362,E2 27727.362} C_VEL
LIN {X 0,Y 578.526,Z 1084.028,A -85,B 0,C 180,E1 27724.659,E2 27724.659} C_VEL
LIN {X 0,Y 579.833,Z 1071.534,A -85,B 0,C 180,E1 27722.273,E2 27722.273} C_VEL
LIN {X 0,Y 581.605,Z 1056.762,A -85,B 0,C 180,E1 27719.803,E2 27719.803} C_VEL
LIN {X 0,Y 583.802,Z 1040,A -85,B 0,C 180,E1 27717.35,E2 27717.35} C_VEL
LIN {X 0,Y 586.283,Z 1022.64,A -85,B 0,C 180,E1 27715.108,E2 27715.108} C_VEL
LIN {X 0,Y 589.172,Z 1003.025,A -85,B 0,C 180,E1 27712.883,E2 27712.883} C_VEL
LIN {X 0,Y 592.245,Z 982.801,A -85,B 0,C 180,E1 27710.868,E2 27710.868} C_VEL
LIN {X 0,Y 595.637,Z 960.564,A -85,B 0,C 180,E1 27708.918,E2 27708.918} C_VEL
LIN {X 0,Y 598.968,Z 938.511,A -85,B 0,C 180,E1 27707.221,E2 27707.221} C_VEL
LIN {X 0,Y 602.313,Z 915.399,A -85,B 0,C 180,E1 27705.679,E2 27705.679} C_VEL
LIN {X 0,Y 605.487,Z 892.182,A -85,B 0,C 180,E1 27704.336,E2 27704.336} C_VEL
LIN {X 0,Y 608.288,Z 870.279,A -85,B 0,C 180,E1 27703.233,E2 27703.233} C_VEL
LIN {X 0,Y 610.736,Z 847.646,A -85,B 0,C 180,E1 27702.271,E2 27702.271} C_VEL
LIN {X 0,Y 613.211,Z 820.912,A -85,B 0,C 180,E1 27701.335,E2 27701.335} C_VEL
LIN {X 0,Y 614.938,Z 797.062,A -85,B 0,C 180,E1 27700.677,E2 27700.677} C_VEL
LIN {X 0,Y 616.186,Z 775.004,A -85,B 0,C 180,E1 27700.2,E2 27700.2} C_VEL
LIN {X 0,Y 617.175,Z 749.954,A -85,B 0,C 180,E1 27699.794,E2 27699.794} C_VEL
LIN {X 0,Y 621.11,Z 573.405,A -85,B 0,C 180,E1 27697.396,E2 27697.396} C_VEL
LIN {X 0,Y 624.963,Z 455.586,A -85,B 0,C 180,E1 27695.671,E2 27695.671} C_VEL
LIN {X 0,Y 626.566,Z 415.779,A -85,B 0,C 180,E1 27695.045,E2 27695.045} C_VEL
LIN {X 0,Y 617.339,Z 400.954,A -85,B 0,C 180,E1 27693.516,E2 27693.516} C_VEL
LIN {X 0,Y 612.097,Z 392.48,A -85,B 0,C 180,E1 27692.423,E2 27692.423} C_VEL
LIN {X 0,Y 608.215,Z 386.286,A -85,B 0,C 180,E1 27691.386,E2 27691.386} C_VEL
LIN {X 0,Y 605.621,Z 381.997,A -85,B 0,C 180,E1 27690.419,E2 27690.419} C_VEL
LIN {X 0,Y 603.679,Z 379.47,A -85,B 0,C 180,E1 27689.216,E2 27689.216} C_VEL
LIN {X 0,Y 603.472,Z 379.346,A -85,B 0,C 180,E1 27688.983,E2 27688.983} C_VEL
LIN {X 0,Y 602.959,Z 380.878,A -85,B 0,C 180,E1 27688.367,E2 27688.367} C_VEL
LIN {X 0,Y 602.985,Z 383.578,A -85,B 0,C 180,E1 27687.615,E2 27687.615} C_VEL
LIN {X 0,Y 604.025,Z 388.928,A -85,B 0,C 180,E1 27686.604,E2 27686.604} C_VEL
LIN {X 0,Y 606.217,Z 396.39,A -85,B 0,C 180,E1 27685.546,E2 27685.546} C_VEL
LIN {X 0,Y 609.096,Z 404.855,A -85,B 0,C 180,E1 27684.629,E2 27684.629} C_VEL
LIN {X 0,Y 614.698,Z 418.969,A -85,B 0,C 180,E1 27683.32,E2 27683.32} C_VEL
LIN {X 0,Y 618.183,Z 425.852,A -85,B 0,C 180,E1 27682.681,E2 27682.681} C_VEL
LIN {X 0,Y 622.689,Z 459.12,A -85,B 0,C 180,E1 27681.435,E2 27681.435} C_VEL
LIN {X 0,Y 625.298,Z 473.889,A -85,B 0,C 180,E1 27680.878,E2 27680.878} C_VEL
LIN {X 0,Y 622.033,Z 584.466,A -85,B 0,C 180,E1 27679.245,E2 27679.245} C_VEL
LIN {X 0,Y 619.343,Z 711.736,A -85,B 0,C 180,E1 27677.494,E2 27677.494} C_VEL
LIN {X 0,Y 616.198,Z 899.35,A -85,B 0,C 180,E1 27675.048,E2 27675.048} C_VEL
LIN {X 0,Y 614.979,Z 927.704,A -85,B 0,C 180,E1 27674.566,E2 27674.566} C_VEL
LIN {X 0,Y 613.254,Z 955.268,A -85,B 0,C 180,E1 27673.919,E2 27673.919} C_VEL
LIN {X 0,Y 611.73,Z 977.148,A -85,B 0,C 180,E1 27673.289,E2 27673.289} C_VEL
LIN {X 0,Y 610.042,Z 998.404,A -85,B 0,C 180,E1 27672.571,E2 27672.571} C_VEL
LIN {X 0,Y 608.471,Z 1016.872,A -85,B 0,C 180,E1 27671.848,E2 27671.848} C_VEL
LIN {X 0,Y 606.744,Z 1032.219,A -85,B 0,C 180,E1 27671.138,E2 27671.138} C_VEL
LIN {X 0,Y 604.013,Z 1052.818,A -85,B 0,C 180,E1 27670.025,E2 27670.025} C_VEL
LIN {X 0,Y 601.264,Z 1072.419,A -85,B 0,C 180,E1 27668.824,E2 27668.824} C_VEL
LIN {X 0,Y 598.197,Z 1093.653,A -85,B 0,C 180,E1 27667.355,E2 27667.355} C_VEL
LIN {X 0,Y 594.742,Z 1116.483,A -85,B 0,C 180,E1 27665.54,E2 27665.54} C_VEL
LIN {X 0,Y 591.984,Z 1134.38,A -85,B 0,C 180,E1 27663.933,E2 27663.933} C_VEL
LIN {X 0,Y 589.483,Z 1150.802,A -85,B 0,C 180,E1 27662.296,E2 27662.296} C_VEL
LIN {X 0,Y 586.784,Z 1168.922,A -85,B 0,C 180,E1 27660.29,E2 27660.29} C_VEL
LIN {X 0,Y 584.179,Z 1187.299,A -85,B 0,C 180,E1 27657.968,E2 27657.968} C_VEL
LIN {X 0,Y 582.266,Z 1201.379,A -85,B 0,C 180,E1 27655.969,E2 27655.969} C_VEL
LIN {X 0,Y 580.623,Z 1214.634,A -85,B 0,C 180,E1 27653.871,E2 27653.871} C_VEL
LIN {X 0,Y 579.016,Z 1229.157,A -85,B 0,C 180,E1 27651.262,E2 27651.262} C_VEL
LIN {X 0,Y 577.946,Z 1240.151,A -85,B 0,C 180,E1 27648.981,E2 27648.981} C_VEL
LIN {X 0,Y 577.208,Z 1249.302,A -85,B 0,C 180,E1 27646.815,E2 27646.815} C_VEL
LIN {X 0,Y 576.681,Z 1257.276,A -85,B 0,C 180,E1 27644.646,E2 27644.646} C_VEL
LIN {X 0,Y 576.272,Z 1265.473,A -85,B 0,C 180,E1 27642.017,E2 27642.017} C_VEL
LIN {X 0,Y 576.004,Z 1272.097,A -85,B 0,C 180,E1 27639.29,E2 27639.29} C_VEL
LIN {X 0,Y 575.954,Z 1276.381,A -85,B 0,C 180,E1 27636.98,E2 27636.98} C_VEL
LIN {X 0,Y 575.916,Z 1279.564,A -85,B 0,C 180,E1 27634.581,E2 27634.581} C_VEL
LIN {X 0,Y 575.91,Z 1281.6,A -85,B 0,C 180,E1 27631.791,E2 27631.791} C_VEL
LIN {X 0,Y 575.865,Z 1281.872,A -85,B 0,C 180,E1 27629.403,E2 27629.403} C_VEL
LIN {X 0,Y 575.907,Z 1281.083,A -85,B 0,C 180,E1 27627.313,E2 27627.313} C_VEL
LIN {X 0,Y 575.919,Z 1279.222,A -85,B 0,C 180,E1 27625.12,E2 27625.12} C_VEL
LIN {X 0,Y 575.963,Z 1276.06,A -85,B 0,C 180,E1 27622.82,E2 27622.82} C_VEL
LIN {X 0,Y 576.034,Z 1271.256,A -85,B 0,C 180,E1 27620.307,E2 27620.307} C_VEL
LIN {X 0,Y 576.311,Z 1264.261,A -85,B 0,C 180,E1 27617.577,E2 27617.577} C_VEL
LIN {X 0,Y 576.715,Z 1256.862,A -85,B 0,C 180,E1 27615.235,E2 27615.235} C_VEL
LIN {X 0,Y 577.236,Z 1248.896,A -85,B 0,C 180,E1 27613.082,E2 27613.082} C_VEL
LIN {X 0,Y 578.042,Z 1239.23,A -85,B 0,C 180,E1 27610.813,E2 27610.813} C_VEL
LIN {X 0,Y 579.359,Z 1225.867,A -85,B 0,C 180,E1 27608.113,E2 27608.113} C_VEL
LIN {X 0,Y 580.813,Z 1212.901,A -85,B 0,C 180,E1 27605.842,E2 27605.842} C_VEL
LIN {X 0,Y 582.457,Z 1199.977,A -85,B 0,C 180,E1 27603.821,E2 27603.821} C_VEL
LIN {X 0,Y 584.737,Z 1183.411,A -85,B 0,C 180,E1 27601.505,E2 27601.505} C_VEL
LIN {X 0,Y 587.334,Z 1165.202,A -85,B 0,C 180,E1 27599.286,E2 27599.286} C_VEL
LIN {X 0,Y 589.714,Z 1149.281,A -85,B 0,C 180,E1 27597.545,E2 27597.545} C_VEL
LIN {X 0,Y 592.341,Z 1132.158,A -85,B 0,C 180,E1 27595.857,E2 27595.857} C_VEL
LIN {X 0,Y 595.736,Z 1109.888,A -85,B 0,C 180,E1 27593.906,E2 27593.906} C_VEL
LIN {X 0,Y 598.812,Z 1089.187,A -85,B 0,C 180,E1 27592.324,E2 27592.324} C_VEL
LIN {X 0,Y 601.605,Z 1069.977,A -85,B 0,C 180,E1 27591.018,E2 27591.018} C_VEL
LIN {X 0,Y 604.642,Z 1048.316,A -85,B 0,C 180,E1 27589.716,E2 27589.716} C_VEL
LIN {X 0,Y 607.727,Z 1024.143,A -85,B 0,C 180,E1 27588.468,E2 27588.468} C_VEL
LIN {X 0,Y 610.197,Z 999.875,A -85,B 0,C 180,E1 27587.442,E2 27587.442} C_VEL
LIN {X 0,Y 612.161,Z 978.997,A -85,B 0,C 180,E1 27586.685,E2 27586.685} C_VEL
LIN {X 0,Y 613.957,Z 957.539,A -85,B 0,C 180,E1 27586.023,E2 27586.023} C_VEL
LIN {X 0,Y 615.696,Z 933.994,A -85,B 0,C 180,E1 27585.428,E2 27585.428} C_VEL
LIN {X 0,Y 617.368,Z 904.368,A -85,B 0,C 180,E1 27584.865,E2 27584.865} C_VEL
LIN {X 0,Y 618.708,Z 854.15,A -85,B 0,C 180,E1 27584.165,E2 27584.165} C_VEL
LIN {X 0,Y 623.428,Z 668.845,A -85,B 0,C 180,E1 27581.591,E2 27581.591} C_VEL
LIN {X 0,Y 627.676,Z 523.008,A -85,B 0,C 180,E1 27579.502,E2 27579.502} C_VEL
LIN {X 0,Y 629.081,Z 473.033,A -85,B 0,C 180,E1 27578.752,E2 27578.752} C_VEL
LIN {X 0,Y 621.082,Z 429.796,A -85,B 0,C 180,E1 27577.021,E2 27577.021} C_VEL
LIN {X 0,Y 612.812,Z 416.934,A -85,B 0,C 180,E1 27575.742,E2 27575.742} C_VEL
LIN {X 0,Y 604.436,Z 399.863,A -85,B 0,C 180,E1 27573.313,E2 27573.313} C_VEL
LIN {X 0,Y 595.734,Z 383.055,A -85,B 0,C 180,E1 27570.68,E2 27570.68} C_VEL
LIN {X 0,Y 587.932,Z 368.812,A -85,B 0,C 180,E1 27568.216,E2 27568.216} C_VEL
LIN {X 0,Y 584.989,Z 363.662,A -85,B 0,C 180,E1 27567.263,E2 27567.263} C_VEL
LIN {X 0,Y 582.461,Z 359.046,A -85,B 0,C 180,E1 27566.399,E2 27566.399} C_VEL
LIN {X 0,Y 580.477,Z 355.609,A -85,B 0,C 180,E1 27565.727,E2 27565.727} C_VEL
LIN {X 0,Y 579.676,Z 354.091,A -85,B 0,C 180,E1 27565.436,E2 27565.436} C_VEL
LIN {X 0,Y 577.664,Z 350.883,A -85,B 0,C 180,E1 27564.764,E2 27564.764} C_VEL
LIN {X 0,Y 577.318,Z 349.481,A -85,B 0,C 180,E1 27564.453,E2 27564.453} C_VEL
LIN {X 0,Y 577.313,Z 349.304,A -85,B 0,C 180,E1 27561.285,E2 27561.285} C_VEL
LIN {X 0,Y 577.294,Z 349.305,A -85,B 0,C 180,E1 27558.035,E2 27558.035} C_VEL
LIN {X 0,Y 577.32,Z 349.303,A -85,B 0,C 180,E1 27554.75,E2 27554.75} C_VEL
LIN {X 0,Y 577.312,Z 349.304,A -85,B 0,C 180,E1 27551.388,E2 27551.388} C_VEL
LIN {X 0,Y 577.291,Z 349.309,A -85,B 0,C 180,E1 27548.065,E2 27548.065} C_VEL
LIN {X 0,Y 577.314,Z 349.301,A -85,B 0,C 180,E1 27544.868,E2 27544.868} C_VEL
LIN {X 0,Y 577.284,Z 349.304,A -85,B 0,C 180,E1 27541.687,E2 27541.687} C_VEL
LIN {X 0,Y 577.319,Z 349.316,A -85,B 0,C 180,E1 27538.511,E2 27538.511} C_VEL
LIN {X 0,Y 577.289,Z 349.315,A -85,B 0,C 180,E1 27535.231,E2 27535.231} C_VEL
LIN {X 0,Y 577.307,Z 349.319,A -85,B 0,C 180,E1 27531.935,E2 27531.935} C_VEL
LIN {X 0,Y 577.308,Z 349.315,A -85,B 0,C 180,E1 27528.713,E2 27528.713} C_VEL
LIN {X 0,Y 577.283,Z 349.319,A -85,B 0,C 180,E1 27525.454,E2 27525.454} C_VEL
LIN {X 0,Y 577.32,Z 349.307,A -85,B 0,C 180,E1 27522.252,E2 27522.252} C_VEL
LIN {X 0,Y 577.275,Z 349.32,A -85,B 0,C 180,E1 27518.989,E2 27518.989} C_VEL
LIN {X 0,Y 577.319,Z 349.312,A -85,B 0,C 180,E1 27515.765,E2 27515.765} C_VEL
LIN {X 0,Y 577.278,Z 349.318,A -85,B 0,C 180,E1 27512.565,E2 27512.565} C_VEL
LIN {X 0,Y 577.295,Z 349.322,A -85,B 0,C 180,E1 27509.212,E2 27509.212} C_VEL
LIN {X 0,Y 577.297,Z 349.316,A -85,B 0,C 180,E1 27506.06,E2 27506.06} C_VEL
LIN {X 0,Y 577.275,Z 349.323,A -85,B 0,C 180,E1 27502.807,E2 27502.807} C_VEL
LIN {X 0,Y 577.318,Z 349.315,A -85,B 0,C 180,E1 27499.645,E2 27499.645} C_VEL
LIN {X 0,Y 577.265,Z 349.322,A -85,B 0,C 180,E1 27496.387,E2 27496.387} C_VEL
LIN {X 0,Y 577.323,Z 349.319,A -85,B 0,C 180,E1 27493.165,E2 27493.165} C_VEL
LIN {X 0,Y 577.261,Z 349.322,A -85,B 0,C 180,E1 27490.039,E2 27490.039} C_VEL
LIN {X 0,Y 577.312,Z 349.321,A -85,B 0,C 180,E1 27486.817,E2 27486.817} C_VEL
LIN {X 0,Y 577.259,Z 349.322,A -85,B 0,C 180,E1 27483.754,E2 27483.754} C_VEL
LIN {X 0,Y 577.296,Z 349.318,A -85,B 0,C 180,E1 27480.496,E2 27480.496} C_VEL
LIN {X 0,Y 577.258,Z 349.32,A -85,B 0,C 180,E1 27477.519,E2 27477.519} C_VEL
LIN {X 0,Y 577.283,Z 349.313,A -85,B 0,C 180,E1 27474.236,E2 27474.236} C_VEL
LIN {X 0,Y 577.254,Z 349.319,A -85,B 0,C 180,E1 27471.33,E2 27471.33} C_VEL
LIN {X 0,Y 577.302,Z 349.313,A -85,B 0,C 180,E1 27468.247,E2 27468.247} C_VEL
LIN {X 0,Y 576.245,Z 349.445,A -85,B 0,C 180,E1 27467.483,E2 27467.483} C_VEL
LIN {X 0,Y 569.822,Z 350.242,A -85,B 0,C 180,E1 27465.337,E2 27465.337} C_VEL
LIN {X 0,Y 569.337,Z 350.302,A -85,B 0,C 180,E1 27464.779,E2 27464.779} C_VEL
LIN {X 0,Y 569.308,Z 350.316,A -85,B 0,C 180,E1 27461.447,E2 27461.447} C_VEL
LIN {X 0,Y 569.372,Z 350.308,A -85,B 0,C 180,E1 27458.279,E2 27458.279} C_VEL
LIN {X 0,Y 569.301,Z 350.306,A -85,B 0,C 180,E1 27455.139,E2 27455.139} C_VEL
LIN {X 0,Y 569.369,Z 350.303,A -85,B 0,C 180,E1 27452.013,E2 27452.013} C_VEL
LIN {X 0,Y 569.296,Z 350.315,A -85,B 0,C 180,E1 27448.893,E2 27448.893} C_VEL
LIN {X 0,Y 569.359,Z 350.29,A -85,B 0,C 180,E1 27445.669,E2 27445.669} C_VEL
LIN {X 0,Y 569.374,Z 350.58,A -85,B 0,C 180,E1 27444.053,E2 27444.053} C_VEL
LIN {X 0,Y 569.915,Z 352.354,A -85,B 0,C 180,E1 27443.768,E2 27443.768} C_VEL
LIN {X 0,Y 571.939,Z 355.254,A -85,B 0,C 180,E1 27443.374,E2 27443.374} C_VEL
LIN {X 0,Y 574.028,Z 357.009,A -85,B 0,C 180,E1 27443.009,E2 27443.009} C_VEL
LIN {X 0,Y 576.457,Z 360.768,A -85,B 0,C 180,E1 27442.55,E2 27442.55} C_VEL
LIN {X 0,Y 578.829,Z 363.071,A -85,B 0,C 180,E1 27442.144,E2 27442.144} C_VEL
LIN {X 0,Y 581.894,Z 367.267,A -85,B 0,C 180,E1 27441.602,E2 27441.602} C_VEL
LIN {X 0,Y 583.798,Z 369.406,A -85,B 0,C 180,E1 27441.282,E2 27441.282} C_VEL
LIN {X 0,Y 587.603,Z 373.903,A -85,B 0,C 180,E1 27440.648,E2 27440.648} C_VEL
LIN {X 0,Y 601.331,Z 391.758,A -85,B 0,C 180,E1 27438.433,E2 27438.433} C_VEL
LIN {X 0,Y 611.971,Z 405.827,A -85,B 0,C 180,E1 27436.856,E2 27436.856} C_VEL
LIN {X 0,Y 622.136,Z 420.387,A -85,B 0,C 180,E1 27435.419,E2 27435.419} C_VEL
LIN {X 0,Y 615.664,Z 625.388,A -85,B 0,C 180,E1 27432.467,E2 27432.467} C_VEL
LIN {X 0,Y 611.827,Z 759.753,A -85,B 0,C 180,E1 27430.572,E2 27430.572} C_VEL
LIN {X 0,Y 610.22,Z 787.81,A -85,B 0,C 180,E1 27430.027,E2 27430.027} C_VEL
LIN {X 0,Y 608.181,Z 813.456,A -85,B 0,C 180,E1 27429.346,E2 27429.346} C_VEL
LIN {X 0,Y 605.915,Z 837.723,A -85,B 0,C 180,E1 27428.549,E2 27428.549} C_VEL
LIN {X 0,Y 602.952,Z 864.244,A -85,B 0,C 180,E1 27427.472,E2 27427.472} C_VEL
LIN {X 0,Y 600.031,Z 886.754,A -85,B 0,C 180,E1 27426.379,E2 27426.379} C_VEL
LIN {X 0,Y 596.641,Z 910.77,A -85,B 0,C 180,E1 27425.019,E2 27425.019} C_VEL
LIN {X 0,Y 593.187,Z 933.768,A -85,B 0,C 180,E1 27423.518,E2 27423.518} C_VEL
LIN {X 0,Y 589.594,Z 956.25,A -85,B 0,C 180,E1 27421.822,E2 27421.822} C_VEL
LIN {X 0,Y 585.993,Z 978.593,A -85,B 0,C 180,E1 27419.895,E2 27419.895} C_VEL
